    movel([-0.101611, -1.453252, -2.511691, -0.747446, 1.570796, 1.469185],accel_mss,speed_ms,0,blend_radius_m)
    movel([-0.098360, -1.448678, -2.515403, -0.748308, 1.570796, 1.472436],accel_mss,speed_ms,0,blend_radius_m)
    movel([-0.092173, -1.439398, -2.522836, -0.750155, 1.570796, 1.478623],accel_mss,speed_ms,0,blend_radius_m)
    movel([-0.087668, -1.432622, -2.528181, -0.751586, 1.570796, 1.483129],accel_mss,speed_ms,0,blend_radius_m)
    movel([-0.083332, -1.426923, -2.532623, -0.752843, 1.570796, 1.487464],accel_mss,speed_ms,0,blend_radius_m)
    movel([-0.078941, -1.421179, -2.537051, -0.754159, 1.570796, 1.491855],accel_mss,speed_ms,0,blend_radius_m)
    movel([-0.091400, -1.427836, -2.531915, -0.752638, 1.570796, 1.479397],accel_mss,speed_ms,0,blend_radius_m)
    movel([-0.097928, -1.431068, -2.529397, -0.751924, 1.570796, 1.472868],accel_mss,speed_ms,0,blend_radius_m)
    movel([-0.104381, -1.433755, -2.527293, -0.751342, 1.570796, 1.466415],accel_mss,speed_ms,0,blend_radius_m)
    movel([-0.107519, -1.434780, -2.526486, -0.751122, 1.570796, 1.463277],accel_mss,speed_ms,0,blend_radius_m)
    movel([-0.110566, -1.435536, -2.525891, -0.750962, 1.570796, 1.460230],accel_mss,speed_ms,0,blend_radius_m)
    movel([-0.113501, -1.435974, -2.525546, -0.750869, 1.570796, 1.457296],accel_mss,speed_ms,0,blend_radius_m)
    movel([-0.116300, -1.436052, -2.525484, -0.750853, 1.570796, 1.454497],accel_mss,speed_ms,0,blend_radius_m)
    movel([-0.118941, -1.435725, -2.525742, -0.750922, 1.570796, 1.451855],accel_mss,speed_ms,0,blend_radius_m)
    movel([-0.121404, -1.434945, -2.526356, -0.751087, 1.570796, 1.449392],accel_mss,speed_ms,0,blend_radius_m)
    movel([-0.123665, -1.433664, -2.527364, -0.751361, 1.570796, 1.447131],accel_mss,speed_ms,0,blend_radius_m)
    movel([-0.125701, -1.431833, -2.528799, -0.751757, 1.570796, 1.445095],accel_mss,speed_ms,0,blend_radius_m)
    movel([-0.127479, -1.429180, -2.530870, -0.752339, 1.570796, 1.443317],accel_mss,speed_ms,0,blend_radius_m)
    movel([-0.128567, -1.425999, -2.533339, -0.753051, 1.570796, 1.442229],accel_mss,speed_ms,0,blend_radius_m)
    movel([-0.128974, -1.422404, -2.536111, -0.753874, 1.570796, 1.441823],accel_mss,speed_ms,0,blend_radius_m)
    movel([-0.128700, -1.418509, -2.539092, -0.754787, 1.570796, 1.442097],accel_mss,speed_ms,0,blend_radius_m)
    movel([-0.127750, -1.414438, -2.542185, -0.755766, 1.570796, 1.443046],accel_mss,speed_ms,0,blend_radius_m)
    movel([-0.126130, -1.410311, -2.545294, -0.756784, 1.570796, 1.444666],accel_mss,speed_ms,0,blend_radius_m)
    movel([-0.123845, -1.406255, -2.548326, -0.757808, 1.570796, 1.446951],accel_mss,speed_ms,0,blend_radius_m)
    movel([-0.120902, -1.402407, -2.551180, -0.758802, 1.570796, 1.449894],accel_mss,speed_ms,0,blend_radius_m)
    movel([-0.118903, -1.400597, -2.552515, -0.759277, 1.570796, 1.451893],accel_mss,speed_ms,0,blend_radius_m)
    movel([-0.116399, -1.398924, -2.553745, -0.759721, 1.570796, 1.454398],accel_mss,speed_ms,0,blend_radius_m)
    movel([-0.114170, -1.397957, -2.554453, -0.759979, 1.570796, 1.456626],accel_mss,speed_ms,0,blend_radius_m)
    movel([-0.113404, -1.397916, -2.554483, -0.759990, 1.570796, 1.457393],accel_mss,speed_ms,0,blend_radius_m)
    movel([-0.113001, -1.398265, -2.554228, -0.759896, 1.570796, 1.457795],accel_mss,speed_ms,0,blend_radius_m)
    movel([-0.114998, -1.399565, -2.553273, -0.759550, 1.570796, 1.455798],accel_mss,speed_ms,0,blend_radius_m)
    movel([-0.116593, -1.400819, -2.552351, -0.759219, 1.570796, 1.454203],accel_mss,speed_ms,0,blend_radius_m)
    movel([-0.117810, -1.402019, -2.551466, -0.758904, 1.570796, 1.452986],accel_mss,speed_ms,0,blend_radius_m)
    movel([-0.118672, -1.403156, -2.550626, -0.758607, 1.570796, 1.452124],accel_mss,speed_ms,0,blend_radius_m)
    movel([-0.119199, -1.404223, -2.549836, -0.758330, 1.570796, 1.451597],accel_mss,speed_ms,0,blend_radius_m)
    movel([-0.119413, -1.405206, -2.549106, -0.758077, 1.570796, 1.451383],accel_mss,speed_ms,0,blend_radius_m)
    movel([-0.119335, -1.406102, -2.548440, -0.757847, 1.570796, 1.451461],accel_mss,speed_ms,0,blend_radius_m)
    movel([-0.118989, -1.406902, -2.547844, -0.757643, 1.570796, 1.451807],accel_mss,speed_ms,0,blend_radius_m)
    movel([-0.117576, -1.408183, -2.546888, -0.757318, 1.570796, 1.453220],accel_mss,speed_ms,0,blend_radius_m)
    movel([-0.115345, -1.408986, -2.546287, -0.757116, 1.570796, 1.455451],accel_mss,speed_ms,0,blend_radius_m)
    movel([-0.112459, -1.409248, -2.546091, -0.757050, 1.570796, 1.458337],accel_mss,speed_ms,0,blend_radius_m)
    movel([-0.109083, -1.408906, -2.546347, -0.757136, 1.570796, 1.461714],accel_mss,speed_ms,0,blend_radius_m)
    movel([-0.106965, -1.408357, -2.546758, -0.757274, 1.570796, 1.463831],accel_mss,speed_ms,0,blend_radius_m)
    movel([-0.104406, -1.407446, -2.547439, -0.757505, 1.570796, 1.466390],accel_mss,speed_ms,0,blend_radius_m)
    movel([-0.098196, -1.404704, -2.549479, -0.758206, 1.570796, 1.472600],accel_mss,speed_ms,0,blend_radius_m)
    movel([-0.090922, -1.401036, -2.552191, -0.759162, 1.570796, 1.479874],accel_mss,speed_ms,0,blend_radius_m)
    movel([-0.083063, -1.396788, -2.555308, -0.760293, 1.570796, 1.487734],accel_mss,speed_ms,0,blend_radius_m)
    movel([-0.067573, -1.387951, -2.561708, -0.762730, 1.570796, 1.503223],accel_mss,speed_ms,0,blend_radius_m)
    movel([-0.055874, -1.381000, -2.566663, -0.764726, 1.570796, 1.514922],accel_mss,speed_ms,0,blend_radius_m)
    movel([-0.049959, -1.377461, -2.569159, -0.765769, 1.570796, 1.520837],accel_mss,speed_ms,0,blend_radius_m)
    movel([-0.046803, -1.375466, -2.570558, -0.766365, 1.570796, 1.523993],accel_mss,speed_ms,0,blend_radius_m)
    movel([-0.044493, -1.373787, -2.571731, -0.766871, 1.570796, 1.526303],accel_mss,speed_ms,0,blend_radius_m)
    movel([-0.043931, -1.373226, -2.572122, -0.767041, 1.570796, 1.526866],accel_mss,speed_ms,0,blend_radius_m)
    movel([-0.043801, -1.372867, -2.572373, -0.767150, 1.570796, 1.526996],accel_mss,speed_ms,0,blend_radius_m)
    movel([-0.044572, -1.372479, -2.572643, -0.767268, 1.570796, 1.526224],accel_mss,speed_ms,0,blend_radius_m)
    movel([-0.047476, -1.372220, -2.572823, -0.767346, 1.570796, 1.523320],accel_mss,speed_ms,0,blend_radius_m)
    movel([-0.050727, -1.372474, -2.572646, -0.767269, 1.570796, 1.520069],accel_mss,speed_ms,0,blend_radius_m)
    movel([-0.057799, -1.373319, -2.572057, -0.767012, 1.570796, 1.512998],accel_mss,speed_ms,0,blend_radius_m)
    movel([-0.061398, -1.373317, -2.572059, -0.767013, 1.570796, 1.509398],accel_mss,speed_ms,0,blend_radius_m)
    movel([-0.064898, -1.372629, -2.572538, -0.767222, 1.570796, 1.505898],accel_mss,speed_ms,0,blend_radius_m)
    movel([-0.066577, -1.371935, -2.573021, -0.767433, 1.570796, 1.504219],accel_mss,speed_ms,0,blend_radius_m)
    movel([-0.068195, -1.370958, -2.573699, -0.767732, 1.570796, 1.502601],accel_mss,speed_ms,0,blend_radius_m)
    movel([-0.069739, -1.369658, -2.574600, -0.768132, 1.570796, 1.501057],accel_mss,speed_ms,0,blend_radius_m)
    movel([-0.071195, -1.367994, -2.575748, -0.768647, 1.570796, 1.499601],accel_mss,speed_ms,0,blend_radius_m)
    movel([-0.072638, -1.365440, -2.577504, -0.769445, 1.570796, 1.498158],accel_mss,speed_ms,0,blend_radius_m)
    movel([-0.073373, -1.362616, -2.579435, -0.770338, 1.570796, 1.497424],accel_mss,speed_ms,0,blend_radius_m)
    movel([-0.073471, -1.359553, -2.581517, -0.771319, 1.570796, 1.497325],accel_mss,speed_ms,0,blend_radius_m)
    movel([-0.073008, -1.356295, -2.583717, -0.772377, 1.570796, 1.497789],accel_mss,speed_ms,0,blend_radius_m)
    movel([-0.072060, -1.352877, -2.586009, -0.773503, 1.570796, 1.498736],accel_mss,speed_ms,0,blend_radius_m)
    movel([-0.070704, -1.349346, -2.588360, -0.774684, 1.570796, 1.500092],accel_mss,speed_ms,0,blend_radius_m)
    movel([-0.069018, -1.345740, -2.590742, -0.775907, 1.570796, 1.501778],accel_mss,speed_ms,0,blend_radius_m)
    movel([-0.067084, -1.342109, -2.593124, -0.777156, 1.570796, 1.503712],accel_mss,speed_ms,0,blend_radius_m)
    movel([-0.062875, -1.335380, -2.597489, -0.779519, 1.570796, 1.507922],accel_mss,speed_ms,0,blend_radius_m)
    movel([-0.058564, -1.329688, -2.601135, -0.781566, 1.570796, 1.512232],accel_mss,speed_ms,0,blend_radius_m)
    movel([-0.054523, -1.325129, -2.604023, -0.783238, 1.570796, 1.516273],accel_mss,speed_ms,0,blend_radius_m)
    movel([-0.051129, -1.321798, -2.606115, -0.784476, 1.570796, 1.519667],accel_mss,speed_ms,0,blend_radius_m)
    movel([-0.045692, -1.317282, -2.608929, -0.786179, 1.570796, 1.525104],accel_mss,speed_ms,0,blend_radius_m)
    movel([-0.040005, -1.313397, -2.611327, -0.787665, 1.570796, 1.530791],accel_mss,speed_ms,0,blend_radius_m)
    movel([-0.034153, -1.310170, -2.613304, -0.788914, 1.570796, 1.536643],accel_mss,speed_ms,0,blend_radius_m)
    movel([-0.028236, -1.307628, -2.614852, -0.789908, 1.570796, 1.542561],accel_mss,speed_ms,0,blend_radius_m)
    movel([-0.022348, -1.305795, -2.615963, -0.790631, 1.570796, 1.548449],accel_mss,speed_ms,0,blend_radius_m)
    movel([-0.016580, -1.304686, -2.616634, -0.791070, 1.570796, 1.554216],accel_mss,speed_ms,0,blend_radius_m)
    movel([-0.011030, -1.304317, -2.616856, -0.791216, 1.570796, 1.559766],accel_mss,speed_ms,0,blend_radius_m)
    movel([-0.005791, -1.304700, -2.616625, -0.791064, 1.570796, 1.565005],accel_mss,speed_ms,0,blend_radius_m)
    movel([-0.001418, -1.305694, -2.616024, -0.790670, 1.570796, 1.569378],accel_mss,speed_ms,0,blend_radius_m)
    movel([0.002673, -1.307080, -2.615185, -0.790124, 1.570796, 1.573469],accel_mss,speed_ms,0,blend_radius_m)
    movel([0.006644, -1.308526, -2.614306, -0.789556, 1.570796, 1.577440],accel_mss,speed_ms,0,blend_radius_m)
    movel([0.010668, -1.309702, -2.613590, -0.789097, 1.570796, 1.581464],accel_mss,speed_ms,0,blend_radius_m)
    movel([0.014918, -1.310286, -2.613234, -0.788870, 1.570796, 1.585715],accel_mss,speed_ms,0,blend_radius_m)
    movel([0.017183, -1.310251, -2.613255, -0.788883, 1.570796, 1.587979],accel_mss,speed_ms,0,blend_radius_m)
    movel([0.019570, -1.309949, -2.613439, -0.789001, 1.570796, 1.590366],accel_mss,speed_ms,0,blend_radius_m)
    movel([0.022104, -1.309335, -2.613814, -0.789240, 1.570796, 1.592900],accel_mss,speed_ms,0,blend_radius_m)
    movel([0.024809, -1.308369, -2.614402, -0.789618, 1.570796, 1.595605],accel_mss,speed_ms,0,blend_radius_m)
    movel([0.027712, -1.307006, -2.615230, -0.790153, 1.570796, 1.598508],accel_mss,speed_ms,0,blend_radius_m)
    movel([0.030836, -1.305204, -2.616321, -0.790864, 1.570796, 1.601633],accel_mss,speed_ms,0,blend_radius_m)
    movel([0.033462, -1.303311, -2.617462, -0.791616, 1.570796, 1.604259],accel_mss,speed_ms,0,blend_radius_m)
    movel([0.035502, -1.301346, -2.618642, -0.792401, 1.570796, 1.606298],accel_mss,speed_ms,0,blend_radius_m)
    movel([0.036986, -1.299357, -2.619831, -0.793201, 1.570796, 1.607782],accel_mss,speed_ms,0,blend_radius_m)
    movel([0.037958, -1.297392, -2.621001, -0.793996, 1.570796, 1.608754],accel_mss,speed_ms,0,blend_radius_m)
    movel([0.038450, -1.295502, -2.622121, -0.794766, 1.570796, 1.609246],accel_mss,speed_ms,0,blend_radius_m)
    movel([0.038495, -1.293743, -2.623160, -0.795486, 1.570796, 1.609292],accel_mss,speed_ms,0,blend_radius_m)
    movel([0.038134, -1.292163, -2.624089, -0.796137, 1.570796, 1.608931],accel_mss,speed_ms,0,blend_radius_m)
    movel([0.037403, -1.290817, -2.624879, -0.796693, 1.570796, 1.608199],accel_mss,speed_ms,0,blend_radius_m)
    movel([0.036339, -1.289760, -2.625497, -0.797132, 1.570796, 1.607135],accel_mss,speed_ms,0,blend_radius_m)
    movel([0.034980, -1.289045, -2.625915, -0.797429, 1.570796, 1.605776],accel_mss,speed_ms,0,blend_radius_m)
    movel([0.033366, -1.288725, -2.626101, -0.797563, 1.570796, 1.604163],accel_mss,speed_ms,0,blend_radius_m)
    movel([0.031539, -1.288853, -2.626027, -0.797510, 1.570796, 1.602335],accel_mss,speed_ms,0,blend_radius_m)
    movel([0.029539, -1.289474, -2.625664, -0.797251, 1.570796, 1.600335],accel_mss,speed_ms,0,blend_radius_m)
    movel([0.027413, -1.290642, -2.624982, -0.796766, 1.570796, 1.598209],accel_mss,speed_ms,0,blend_radius_m)
    movel([0.025201, -1.292403, -2.623948, -0.796037, 1.570796, 1.595998],accel_mss,speed_ms,0,blend_radius_m)
    movel([0.022949, -1.294798, -2.622537, -0.795054, 1.570796, 1.593746],accel_mss,speed_ms,0,blend_radius_m)
    movel([0.024835, -1.294234, -2.622870, -0.795285, 1.570796, 1.595631],accel_mss,speed_ms,0,blend_radius_m)
    movel([0.026385, -1.294077, -2.622963, -0.795349, 1.570796, 1.597182],accel_mss,speed_ms,0,blend_radius_m)
    movel([0.027564, -1.294304, -2.622829, -0.795256, 1.570796, 1.598361],accel_mss,speed_ms,0,blend_radius_m)
    movel([0.028342, -1.294888, -2.622484, -0.795017, 1.570796, 1.599138],accel_mss,speed_ms,0,blend_radius_m)
    movel([0.028683, -1.295809, -2.621940, -0.794641, 1.570796, 1.599479],accel_mss,speed_ms,0,blend_radius_m)
    movel([0.028557, -1.297039, -2.621210, -0.794140, 1.570796, 1.599354],accel_mss,speed_ms,0,blend_radius_m)
    movel([0.027935, -1.298550, -2.620312, -0.793527, 1.570796, 1.598731],accel_mss,speed_ms,0,blend_radius_m)
    movel([0.026784, -1.300320, -2.619256, -0.792813, 1.570796, 1.597581],accel_mss,speed_ms,0,blend_radius_m)
    movel([0.024280, -1.303118, -2.617578, -0.791693, 1.570796, 1.595077],accel_mss,speed_ms,0,blend_radius_m)
    movel([0.021602, -1.305191, -2.616329, -0.790870, 1.570796, 1.592398],accel_mss,speed_ms,0,blend_radius_m)
    movel([0.018815, -1.306593, -2.615480, -0.790316, 1.570796, 1.589612],accel_mss,speed_ms,0,blend_radius_m)
    movel([0.016000, -1.307372, -2.615008, -0.790009, 1.570796, 1.586796],accel_mss,speed_ms,0,blend_radius_m)
    movel([0.013225, -1.307572, -2.614887, -0.789931, 1.570796, 1.584021],accel_mss,speed_ms,0,blend_radius_m)
    movel([0.010566, -1.307233, -2.615092, -0.790064, 1.570796, 1.581362],accel_mss,speed_ms,0,blend_radius_m)
    movel([0.008102, -1.306397, -2.615599, -0.790393, 1.570796, 1.578898],accel_mss,speed_ms,0,blend_radius_m)
    movel([0.005906, -1.305103, -2.616381, -0.790904, 1.570796, 1.576702],accel_mss,speed_ms,0,blend_radius_m)
    movel([0.004062, -1.303381, -2.617420, -0.791588, 1.570796, 1.574859],accel_mss,speed_ms,0,blend_radius_m)
    movel([0.002647, -1.301272, -2.618686, -0.792431, 1.570796, 1.573443],accel_mss,speed_ms,0,blend_radius_m)
    movel([0.001748, -1.298803, -2.620161, -0.793425, 1.570796, 1.572545],accel_mss,speed_ms,0,blend_radius_m)
    movel([0.001450, -1.296012, -2.621819, -0.794558, 1.570796, 1.572246],accel_mss,speed_ms,0,blend_radius_m)
    movel([0.001841, -1.292927, -2.623641, -0.795822, 1.570796, 1.572637],accel_mss,speed_ms,0,blend_radius_m)
    movel([0.003010, -1.289582, -2.625601, -0.797206, 1.570796, 1.573806],accel_mss,speed_ms,0,blend_radius_m)
    movel([0.005052, -1.286011, -2.627679, -0.798699, 1.570796, 1.575848],accel_mss,speed_ms,0,blend_radius_m)
    movel([0.008055, -1.282252, -2.629848, -0.800289, 1.570796, 1.578851],accel_mss,speed_ms,0,blend_radius_m)
    movel([0.010545, -1.279696, -2.631313, -0.801380, 1.570796, 1.581341],accel_mss,speed_ms,0,blend_radius_m)
    movel([0.013182, -1.277305, -2.632676, -0.802408, 1.570796, 1.583978],accel_mss,speed_ms,0,blend_radius_m)
    movel([0.015934, -1.275092, -2.633932, -0.803365, 1.570796, 1.586731],accel_mss,speed_ms,0,blend_radius_m)
    movel([0.018783, -1.273077, -2.635069, -0.804243, 1.570796, 1.589579],accel_mss,speed_ms,0,blend_radius_m)
    movel([0.021695, -1.271275, -2.636082, -0.805032, 1.570796, 1.592491],accel_mss,speed_ms,0,blend_radius_m)
    movel([0.024648, -1.269703, -2.636963, -0.805723, 1.570796, 1.595444],accel_mss,speed_ms,0,blend_radius_m)
    movel([0.027613, -1.268378, -2.637703, -0.806308, 1.570796, 1.598410],accel_mss,speed_ms,0,blend_radius_m)
    movel([0.030563, -1.267314, -2.638295, -0.806780, 1.570796, 1.601360],accel_mss,speed_ms,0,blend_radius_m)
    movel([0.033469, -1.266531, -2.638731, -0.807128, 1.570796, 1.604266],accel_mss,speed_ms,0,blend_radius_m)
    movel([0.036305, -1.266038, -2.639004, -0.807347, 1.570796, 1.607101],accel_mss,speed_ms,0,blend_radius_m)
    movel([0.039042, -1.265856, -2.639105, -0.807428, 1.570796, 1.609838],accel_mss,speed_ms,0,blend_radius_m)
    movel([0.041654, -1.265996, -2.639027, -0.807366, 1.570796, 1.612451],accel_mss,speed_ms,0,blend_radius_m)
    movel([0.044111, -1.266472, -2.638763, -0.807154, 1.570796, 1.614907],accel_mss,speed_ms,0,blend_radius_m)
    movel([0.046390, -1.267293, -2.638307, -0.806789, 1.570796, 1.617186],accel_mss,speed_ms,0,blend_radius_m)
    movel([0.048461, -1.268477, -2.637648, -0.806264, 1.570796, 1.619257],accel_mss,speed_ms,0,blend_radius_m)
    movel([0.050299, -1.270031, -2.636779, -0.805578, 1.570796, 1.621095],accel_mss,speed_ms,0,blend_radius_m)
    movel([0.051489, -1.272144, -2.635594, -0.804650, 1.570796, 1.622286],accel_mss,speed_ms,0,blend_radius_m)
    movel([0.052205, -1.274852, -2.634067, -0.803469, 1.570796, 1.623002],accel_mss,speed_ms,0,blend_radius_m)
    movel([0.052659, -1.277284, -2.632688, -0.802416, 1.570796, 1.623456],accel_mss,speed_ms,0,blend_radius_m)
    movel([0.053064, -1.278582, -2.631949, -0.801858, 1.570796, 1.623860],accel_mss,speed_ms,0,blend_radius_m)
    movel([0.054264, -1.278779, -2.631837, -0.801773, 1.570796, 1.625060],accel_mss,speed_ms,0,blend_radius_m)
    movel([0.056461, -1.278666, -2.631901, -0.801821, 1.570796, 1.627257],accel_mss,speed_ms,0,blend_radius_m)
    movel([0.058885, -1.278544, -2.631971, -0.801874, 1.570796, 1.629681],accel_mss,speed_ms,0,blend_radius_m)
    movel([0.060765, -1.278700, -2.631882, -0.801807, 1.570796, 1.631562],accel_mss,speed_ms,0,blend_radius_m)
    movel([0.062834, -1.279532, -2.631407, -0.801450, 1.570796, 1.633631],accel_mss,speed_ms,0,blend_radius_m)
    movel([0.064472, -1.280680, -2.630751, -0.800959, 1.570796, 1.635268],accel_mss,speed_ms,0,blend_radius_m)
    movel([0.065692, -1.282108, -2.629931, -0.800350, 1.570796, 1.636488],accel_mss,speed_ms,0,blend_radius_m)
    movel([0.066513, -1.283776, -2.628971, -0.799642, 1.570796, 1.637309],accel_mss,speed_ms,0,blend_radius_m)
    movel([0.066955, -1.285648, -2.627889, -0.798852, 1.570796, 1.637752],accel_mss,speed_ms,0,blend_radius_m)
    movel([0.067036, -1.287682, -2.626708, -0.797998, 1.570796, 1.637832],accel_mss,speed_ms,0,blend_radius_m)
    movel([0.066776, -1.289843, -2.625448, -0.797097, 1.570796, 1.637572],accel_mss,speed_ms,0,blend_radius_m)
    movel([0.066191, -1.292094, -2.624130, -0.796165, 1.570796, 1.636988],accel_mss,speed_ms,0,blend_radius_m)
    movel([0.065300, -1.294401, -2.622772, -0.795216, 1.570796, 1.636097],accel_mss,speed_ms,0,blend_radius_m)
    movel([0.064122, -1.296725, -2.621397, -0.794267, 1.570796, 1.634918],accel_mss,speed_ms,0,blend_radius_m)
    movel([0.062673, -1.299035, -2.620023, -0.793331, 1.570796, 1.633469],accel_mss,speed_ms,0,blend_radius_m)
    speed_ms = 0.003
    movel([0.062673, -1.292173, -2.616738, -0.803478, 1.570796, 1.633469],accel_mss,speed_ms,0,blend_radius_m)
    speed_ms = 0.05
    movel([0.062673, -1.265901, -2.603322, -0.843166, 1.570796, 1.633469],accel_mss,speed_ms,0,blend_radius_m)
    #M_RunCode9
    movel([0.079276, -1.257744, -2.607923, -0.846722, 1.570796, 1.650073],accel_mss,speed_ms,0,blend_radius_m)
    #M_RunCode3
    movel([0.079276, -1.284127, -2.621447, -0.806816, 1.570796, 1.650073],accel_mss,speed_ms,0,blend_radius_m)
    speed_ms = 0.003
    movel([0.079276, -1.291022, -2.624759, -0.796608, 1.570796, 1.650073],accel_mss,speed_ms,0,blend_radius_m)
    speed_ms = 0.02
    movel([0.079182, -1.289313, -2.625758, -0.797318, 1.570796, 1.649979],accel_mss,speed_ms,0,blend_radius_m)
    movel([0.079578, -1.285585, -2.627926, -0.798879, 1.570796, 1.650374],accel_mss,speed_ms,0,blend_radius_m)
    movel([0.079753, -1.282031, -2.629975, -0.800383, 1.570796, 1.650549],accel_mss,speed_ms,0,blend_radius_m)
    movel([0.079381, -1.280546, -2.630827, -0.801016, 1.570796, 1.650178],accel_mss,speed_ms,0,blend_radius_m)
    movel([0.078497, -1.279378, -2.631495, -0.801516, 1.570796, 1.649293],accel_mss,speed_ms,0,blend_radius_m)
    movel([0.079533, -1.279857, -2.631221, -0.801311, 1.570796, 1.650329],accel_mss,speed_ms,0,blend_radius_m)
    movel([0.081004, -1.281148, -2.630482, -0.800759, 1.570796, 1.651801],accel_mss,speed_ms,0,blend_radius_m)
    movel([0.081818, -1.282779, -2.629545, -0.800065, 1.570796, 1.652614],accel_mss,speed_ms,0,blend_radius_m)
    movel([0.082178, -1.284645, -2.628469, -0.799275, 1.570796, 1.652974],accel_mss,speed_ms,0,blend_radius_m)
    movel([0.082289, -1.286641, -2.627313, -0.798435, 1.570796, 1.653085],accel_mss,speed_ms,0,blend_radius_m)
    movel([0.082574, -1.290622, -2.624993, -0.796774, 1.570796, 1.653370],accel_mss,speed_ms,0,blend_radius_m)
    movel([0.083146, -1.292412, -2.623943, -0.796034, 1.570796, 1.653942],accel_mss,speed_ms,0,blend_radius_m)
    movel([0.084268, -1.293936, -2.623046, -0.795407, 1.570796, 1.655064],accel_mss,speed_ms,0,blend_radius_m)
    movel([0.086018, -1.295241, -2.622276, -0.794873, 1.570796, 1.656814],accel_mss,speed_ms,0,blend_radius_m)
    movel([0.087065, -1.295825, -2.621930, -0.794634, 1.570796, 1.657861],accel_mss,speed_ms,0,blend_radius_m)
    movel([0.087819, -1.295990, -2.621832, -0.794567, 1.570796, 1.658615],accel_mss,speed_ms,0,blend_radius_m)
    movel([0.089062, -1.295029, -2.622401, -0.794959, 1.570796, 1.659858],accel_mss,speed_ms,0,blend_radius_m)
    movel([0.090104, -1.294278, -2.622844, -0.795267, 1.570796, 1.660900],accel_mss,speed_ms,0,blend_radius_m)
    movel([0.091245, -1.293667, -2.623204, -0.795517, 1.570796, 1.662041],accel_mss,speed_ms,0,blend_radius_m)
    movel([0.093544, -1.292886, -2.623664, -0.795839, 1.570796, 1.664341],accel_mss,speed_ms,0,blend_radius_m)
    movel([0.095252, -1.292611, -2.623826, -0.795952, 1.570796, 1.666049],accel_mss,speed_ms,0,blend_radius_m)
    movel([0.096505, -1.292746, -2.623747, -0.795896, 1.570796, 1.667301],accel_mss,speed_ms,0,blend_radius_m)
    movel([0.097444, -1.293201, -2.623479, -0.795709, 1.570796, 1.668240],accel_mss,speed_ms,0,blend_radius_m)
    movel([0.098946, -1.294696, -2.622598, -0.795095, 1.570796, 1.669743],accel_mss,speed_ms,0,blend_radius_m)
    movel([0.100895, -1.296364, -2.621610, -0.794414, 1.570796, 1.671692],accel_mss,speed_ms,0,blend_radius_m)
    movel([0.104110, -1.298008, -2.620635, -0.793747, 1.570796, 1.674906],accel_mss,speed_ms,0,blend_radius_m)
    movel([0.107423, -1.299511, -2.619739, -0.793139, 1.570796, 1.678219],accel_mss,speed_ms,0,blend_radius_m)
    movel([0.110560, -1.301203, -2.618727, -0.792458, 1.570796, 1.681356],accel_mss,speed_ms,0,blend_radius_m)
    movel([0.113253, -1.303396, -2.617411, -0.791582, 1.570796, 1.684050],accel_mss,speed_ms,0,blend_radius_m)
    movel([0.114384, -1.304882, -2.616515, -0.790992, 1.570796, 1.685180],accel_mss,speed_ms,0,blend_radius_m)
    movel([0.115256, -1.306555, -2.615503, -0.790331, 1.570796, 1.686053],accel_mss,speed_ms,0,blend_radius_m)
    movel([0.116468, -1.310252, -2.613254, -0.788883, 1.570796, 1.687264],accel_mss,speed_ms,0,blend_radius_m)
    movel([0.117372, -1.314078, -2.610908, -0.787403, 1.570796, 1.688168],accel_mss,speed_ms,0,blend_radius_m)
    movel([0.118449, -1.317628, -2.608714, -0.786047, 1.570796, 1.689246],accel_mss,speed_ms,0,blend_radius_m)
    movel([0.121104, -1.322927, -2.605407, -0.784054, 1.570796, 1.691901],accel_mss,speed_ms,0,blend_radius_m)
    movel([0.122316, -1.325141, -2.604015, -0.783233, 1.570796, 1.693112],accel_mss,speed_ms,0,blend_radius_m)
    movel([0.123257, -1.327360, -2.602613, -0.782416, 1.570796, 1.694054],accel_mss,speed_ms,0,blend_radius_m)
    movel([0.123798, -1.329795, -2.601066, -0.781528, 1.570796, 1.694594],accel_mss,speed_ms,0,blend_radius_m)
    movel([0.123793, -1.332661, -2.599236, -0.780492, 1.570796, 1.694590],accel_mss,speed_ms,0,blend_radius_m)
    movel([0.123109, -1.336167, -2.596982, -0.779240, 1.570796, 1.693905],accel_mss,speed_ms,0,blend_radius_m)
    movel([0.121617, -1.340512, -2.594165, -0.777711, 1.570796, 1.692413],accel_mss,speed_ms,0,blend_radius_m)
    movel([0.120010, -1.344054, -2.591850, -0.776485, 1.570796, 1.690807],accel_mss,speed_ms,0,blend_radius_m)
    movel([0.118181, -1.347275, -2.589730, -0.775384, 1.570796, 1.688977],accel_mss,speed_ms,0,blend_radius_m)
    movel([0.116146, -1.350191, -2.587799, -0.774399, 1.570796, 1.686942],accel_mss,speed_ms,0,blend_radius_m)
    movel([0.113919, -1.352822, -2.586045, -0.773521, 1.570796, 1.684715],accel_mss,speed_ms,0,blend_radius_m)
    movel([0.111524, -1.355182, -2.584465, -0.772742, 1.570796, 1.682320],accel_mss,speed_ms,0,blend_radius_m)
    movel([0.108974, -1.357288, -2.583048, -0.772053, 1.570796, 1.679770],accel_mss,speed_ms,0,blend_radius_m)
    movel([0.106287, -1.359152, -2.581788, -0.771448, 1.570796, 1.677084],accel_mss,speed_ms,0,blend_radius_m)
    movel([0.103479, -1.360792, -2.580676, -0.770920, 1.570796, 1.674275],accel_mss,speed_ms,0,blend_radius_m)
    movel([0.100570, -1.362219, -2.579706, -0.770464, 1.570796, 1.671366],accel_mss,speed_ms,0,blend_radius_m)
    movel([0.097571, -1.363450, -2.578866, -0.770073, 1.570796, 1.668367],accel_mss,speed_ms,0,blend_radius_m)
    movel([0.091375, -1.365371, -2.577552, -0.769466, 1.570796, 1.662171],accel_mss,speed_ms,0,blend_radius_m)
    movel([0.085030, -1.366656, -2.576669, -0.769064, 1.570796, 1.655826],accel_mss,speed_ms,0,blend_radius_m)
    movel([0.078670, -1.367404, -2.576155, -0.768830, 1.570796, 1.649466],accel_mss,speed_ms,0,blend_radius_m)
    movel([0.072831, -1.367616, -2.576008, -0.768764, 1.570796, 1.643627],accel_mss,speed_ms,0,blend_radius_m)
    movel([0.065389, -1.367790, -2.575889, -0.768710, 1.570796, 1.636186],accel_mss,speed_ms,0,blend_radius_m)
    movel([0.057017, -1.368376, -2.575485, -0.768528, 1.570796, 1.627813],accel_mss,speed_ms,0,blend_radius_m)
    movel([0.052698, -1.368956, -2.575085, -0.768348, 1.570796, 1.623495],accel_mss,speed_ms,0,blend_radius_m)
    movel([0.048406, -1.369796, -2.574504, -0.768089, 1.570796, 1.619202],accel_mss,speed_ms,0,blend_radius_m)
    movel([0.044238, -1.370942, -2.573710, -0.767737, 1.570796, 1.615034],accel_mss,speed_ms,0,blend_radius_m)
    movel([0.040279, -1.372440, -2.572669, -0.767279, 1.570796, 1.611075],accel_mss,speed_ms,0,blend_radius_m)
    movel([0.036623, -1.374335, -2.571349, -0.766705, 1.570796, 1.607420],accel_mss,speed_ms,0,blend_radius_m)
    movel([0.033366, -1.376665, -2.569718, -0.766006, 1.570796, 1.604162],accel_mss,speed_ms,0,blend_radius_m)
    movel([0.031912, -1.378007, -2.568775, -0.765607, 1.570796, 1.602708],accel_mss,speed_ms,0,blend_radius_m)
    movel([0.030592, -1.379474, -2.567741, -0.765174, 1.570796, 1.601389],accel_mss,speed_ms,0,blend_radius_m)
    movel([0.029416, -1.381068, -2.566615, -0.764706, 1.570796, 1.600212],accel_mss,speed_ms,0,blend_radius_m)
    movel([0.028394, -1.382796, -2.565389, -0.764204, 1.570796, 1.599190],accel_mss,speed_ms,0,blend_radius_m)
    movel([0.027538, -1.384663, -2.564061, -0.763666, 1.570796, 1.598334],accel_mss,speed_ms,0,blend_radius_m)
    movel([0.026856, -1.386673, -2.562624, -0.763092, 1.570796, 1.597652],accel_mss,speed_ms,0,blend_radius_m)
    movel([0.026061, -1.391141, -2.559411, -0.761837, 1.570796, 1.596857],accel_mss,speed_ms,0,blend_radius_m)
    movel([0.026322, -1.393089, -2.558001, -0.761299, 1.570796, 1.597118],accel_mss,speed_ms,0,blend_radius_m)
    movel([0.027050, -1.394855, -2.556718, -0.760816, 1.570796, 1.597846],accel_mss,speed_ms,0,blend_radius_m)
    movel([0.028269, -1.396415, -2.555581, -0.760393, 1.570796, 1.599066],accel_mss,speed_ms,0,blend_radius_m)
    movel([0.029998, -1.397736, -2.554615, -0.760038, 1.570796, 1.600794],accel_mss,speed_ms,0,blend_radius_m)
    movel([0.031257, -1.394714, -2.556821, -0.760855, 1.570796, 1.602054],accel_mss,speed_ms,0,blend_radius_m)
    movel([0.032818, -1.391796, -2.558938, -0.761656, 1.570796, 1.603614],accel_mss,speed_ms,0,blend_radius_m)
    movel([0.034657, -1.389000, -2.560954, -0.762435, 1.570796, 1.605453],accel_mss,speed_ms,0,blend_radius_m)
    movel([0.036750, -1.386344, -2.562860, -0.763185, 1.570796, 1.607546],accel_mss,speed_ms,0,blend_radius_m)
    movel([0.039067, -1.383848, -2.564641, -0.763900, 1.570796, 1.609864],accel_mss,speed_ms,0,blend_radius_m)
    movel([0.041589, -1.381528, -2.566289, -0.764572, 1.570796, 1.612385],accel_mss,speed_ms,0,blend_radius_m)
    movel([0.044286, -1.379407, -2.567789, -0.765193, 1.570796, 1.615082],accel_mss,speed_ms,0,blend_radius_m)
    movel([0.047131, -1.377502, -2.569130, -0.765757, 1.570796, 1.617927],accel_mss,speed_ms,0,blend_radius_m)
    movel([0.050098, -1.375832, -2.570302, -0.766255, 1.570796, 1.620894],accel_mss,speed_ms,0,blend_radius_m)
    movel([0.053153, -1.374420, -2.571289, -0.766679, 1.570796, 1.623949],accel_mss,speed_ms,0,blend_radius_m)
    movel([0.056273, -1.373281, -2.572084, -0.767024, 1.570796, 1.627069],accel_mss,speed_ms,0,blend_radius_m)
    movel([0.059427, -1.372434, -2.572674, -0.767281, 1.570796, 1.630223],accel_mss,speed_ms,0,blend_radius_m)
    movel([0.062582, -1.371902, -2.573043, -0.767443, 1.570796, 1.633378],accel_mss,speed_ms,0,blend_radius_m)
    movel([0.065712, -1.371700, -2.573184, -0.767505, 1.570796, 1.636508],accel_mss,speed_ms,0,blend_radius_m)
    movel([0.068788, -1.371845, -2.573083, -0.767461, 1.570796, 1.639584],accel_mss,speed_ms,0,blend_radius_m)
    movel([0.071774, -1.372351, -2.572731, -0.767306, 1.570796, 1.642571],accel_mss,speed_ms,0,blend_radius_m)
    movel([0.074076, -1.373042, -2.572251, -0.767097, 1.570796, 1.644873],accel_mss,speed_ms,0,blend_radius_m)
    movel([0.076126, -1.373943, -2.571622, -0.766823, 1.570796, 1.646923],accel_mss,speed_ms,0,blend_radius_m)
    movel([0.077925, -1.375042, -2.570854, -0.766492, 1.570796, 1.648722],accel_mss,speed_ms,0,blend_radius_m)
    movel([0.079482, -1.376320, -2.569960, -0.766109, 1.570796, 1.650279],accel_mss,speed_ms,0,blend_radius_m)
    movel([0.081892, -1.379341, -2.567836, -0.765213, 1.570796, 1.652688],accel_mss,speed_ms,0,blend_radius_m)
    movel([0.083393, -1.382869, -2.565338, -0.764183, 1.570796, 1.654189],accel_mss,speed_ms,0,blend_radius_m)
    movel([0.084042, -1.386769, -2.562555, -0.763064, 1.570796, 1.654838],accel_mss,speed_ms,0,blend_radius_m)
    movel([0.083884, -1.390908, -2.559579, -0.761902, 1.570796, 1.654680],accel_mss,speed_ms,0,blend_radius_m)
    movel([0.082968, -1.395161, -2.556495, -0.760733, 1.570796, 1.653765],accel_mss,speed_ms,0,blend_radius_m)
    movel([0.081349, -1.399402, -2.553394, -0.759594, 1.570796, 1.652145],accel_mss,speed_ms,0,blend_radius_m)
    movel([0.079067, -1.403514, -2.550361, -0.758514, 1.570796, 1.649863],accel_mss,speed_ms,0,blend_radius_m)
    movel([0.076168, -1.407383, -2.547485, -0.757521, 1.570796, 1.646964],accel_mss,speed_ms,0,blend_radius_m)
    movel([0.072694, -1.410900, -2.544852, -0.756637, 1.570796, 1.643491],accel_mss,speed_ms,0,blend_radius_m)
    movel([0.070752, -1.412493, -2.543653, -0.756243, 1.570796, 1.641548],accel_mss,speed_ms,0,blend_radius_m)
    movel([0.068679, -1.413959, -2.542547, -0.755883, 1.570796, 1.639476],accel_mss,speed_ms,0,blend_radius_m)
    movel([0.066479, -1.415283, -2.541545, -0.755561, 1.570796, 1.637275],accel_mss,speed_ms,0,blend_radius_m)
    movel([0.064155, -1.416455, -2.540656, -0.755278, 1.570796, 1.634951],accel_mss,speed_ms,0,blend_radius_m)
    movel([0.061709, -1.417461, -2.539891, -0.755037, 1.570796, 1.632505],accel_mss,speed_ms,0,blend_radius_m)
    movel([0.059146, -1.418290, -2.539259, -0.754840, 1.570796, 1.629943],accel_mss,speed_ms,0,blend_radius_m)
    movel([0.056468, -1.418926, -2.538774, -0.754689, 1.570796, 1.627265],accel_mss,speed_ms,0,blend_radius_m)
    movel([0.053678, -1.419360, -2.538443, -0.754586, 1.570796, 1.624474],accel_mss,speed_ms,0,blend_radius_m)
    movel([0.050775, -1.419580, -2.538275, -0.754534, 1.570796, 1.621571],accel_mss,speed_ms,0,blend_radius_m)
    movel([0.047763, -1.419572, -2.538281, -0.754536, 1.570796, 1.618560],accel_mss,speed_ms,0,blend_radius_m)
    movel([0.045463, -1.419231, -2.538541, -0.754617, 1.570796, 1.616260],accel_mss,speed_ms,0,blend_radius_m)
    movel([0.039389, -1.417785, -2.539644, -0.754960, 1.570796, 1.610185],accel_mss,speed_ms,0,blend_radius_m)
    movel([0.035310, -1.416454, -2.540656, -0.755279, 1.570796, 1.606106],accel_mss,speed_ms,0,blend_radius_m)
    movel([0.030735, -1.414611, -2.542054, -0.755724, 1.570796, 1.601531],accel_mss,speed_ms,0,blend_radius_m)
    movel([0.025805, -1.412176, -2.543892, -0.756321, 1.570796, 1.596601],accel_mss,speed_ms,0,blend_radius_m)
    movel([0.020668, -1.409061, -2.546231, -0.757097, 1.570796, 1.591464],accel_mss,speed_ms,0,blend_radius_m)
    movel([0.017364, -1.406564, -2.548096, -0.757729, 1.570796, 1.588160],accel_mss,speed_ms,0,blend_radius_m)
    movel([0.014706, -1.403978, -2.550018, -0.758394, 1.570796, 1.585503],accel_mss,speed_ms,0,blend_radius_m)
    movel([0.012640, -1.401332, -2.551973, -0.759084, 1.570796, 1.583436],accel_mss,speed_ms,0,blend_radius_m)
    movel([0.011109, -1.398658, -2.553940, -0.759792, 1.570796, 1.581905],accel_mss,speed_ms,0,blend_radius_m)
    movel([0.010057, -1.395981, -2.555897, -0.760510, 1.570796, 1.580853],accel_mss,speed_ms,0,blend_radius_m)
    movel([0.009421, -1.393343, -2.557817, -0.761229, 1.570796, 1.580217],accel_mss,speed_ms,0,blend_radius_m)
    movel([0.009147, -1.390773, -2.559676, -0.761939, 1.570796, 1.579944],accel_mss,speed_ms,0,blend_radius_m)
    movel([0.009172, -1.388310, -2.561450, -0.762629, 1.570796, 1.579968],accel_mss,speed_ms,0,blend_radius_m)
    movel([0.009872, -1.383854, -2.564637, -0.763898, 1.570796, 1.580668],accel_mss,speed_ms,0,blend_radius_m)
    movel([0.011015, -1.380280, -2.567172, -0.764937, 1.570796, 1.581812],accel_mss,speed_ms,0,blend_radius_m)
    movel([0.012088, -1.377904, -2.568847, -0.765637, 1.570796, 1.582885],accel_mss,speed_ms,0,blend_radius_m)
    movel([0.012563, -1.377043, -2.569453, -0.765893, 1.570796, 1.583360],accel_mss,speed_ms,0,blend_radius_m)
    movel([0.015106, -1.373061, -2.572237, -0.767091, 1.570796, 1.585902],accel_mss,speed_ms,0,blend_radius_m)
    movel([0.017908, -1.369437, -2.574752, -0.768200, 1.570796, 1.588704],accel_mss,speed_ms,0,blend_radius_m)
    movel([0.020922, -1.366164, -2.577007, -0.769218, 1.570796, 1.591718],accel_mss,speed_ms,0,blend_radius_m)
    movel([0.024100, -1.363226, -2.579019, -0.770144, 1.570796, 1.594896],accel_mss,speed_ms,0,blend_radius_m)
    movel([0.027388, -1.360613, -2.580798, -0.770978, 1.570796, 1.598185],accel_mss,speed_ms,0,blend_radius_m)
    movel([0.030737, -1.358314, -2.582355, -0.771720, 1.570796, 1.601534],accel_mss,speed_ms,0,blend_radius_m)
    movel([0.034100, -1.356306, -2.583709, -0.772374, 1.570796, 1.604897],accel_mss,speed_ms,0,blend_radius_m)
    movel([0.037421, -1.354581, -2.584868, -0.772940, 1.570796, 1.608218],accel_mss,speed_ms,0,blend_radius_m)
    movel([0.043743, -1.351902, -2.586660, -0.773827, 1.570796, 1.614539],accel_mss,speed_ms,0,blend_radius_m)
    movel([0.049305, -1.350125, -2.587843, -0.774422, 1.570796, 1.620101],accel_mss,speed_ms,0,blend_radius_m)
    movel([0.053716, -1.349086, -2.588532, -0.774771, 1.570796, 1.624512],accel_mss,speed_ms,0,blend_radius_m)
    movel([0.056596, -1.348614, -2.588845, -0.774930, 1.570796, 1.627392],accel_mss,speed_ms,0,blend_radius_m)
    movel([0.063455, -1.347440, -2.589622, -0.775328, 1.570796, 1.634252],accel_mss,speed_ms,0,blend_radius_m)
    movel([0.070821, -1.346624, -2.590160, -0.775605, 1.570796, 1.641617],accel_mss,speed_ms,0,blend_radius_m)
    movel([0.078298, -1.345957, -2.590600, -0.775832, 1.570796, 1.649094],accel_mss,speed_ms,0,blend_radius_m)
    movel([0.085507, -1.345214, -2.591089, -0.776087, 1.570796, 1.656303],accel_mss,speed_ms,0,blend_radius_m)
    movel([0.092080, -1.344157, -2.591783, -0.776449, 1.570796, 1.662876],accel_mss,speed_ms,0,blend_radius_m)
    movel([0.095014, -1.343433, -2.592257, -0.776698, 1.570796, 1.665810],accel_mss,speed_ms,0,blend_radius_m)
    movel([0.097652, -1.342538, -2.592843, -0.777007, 1.570796, 1.668448],accel_mss,speed_ms,0,blend_radius_m)
    movel([0.099954, -1.341436, -2.593563, -0.777390, 1.570796, 1.670750],accel_mss,speed_ms,0,blend_radius_m)
    movel([0.101868, -1.340096, -2.594436, -0.777857, 1.570796, 1.672665],accel_mss,speed_ms,0,blend_radius_m)
    movel([0.103355, -1.338484, -2.595484, -0.778422, 1.570796, 1.674151],accel_mss,speed_ms,0,blend_radius_m)
    movel([0.104366, -1.336568, -2.596724, -0.779098, 1.570796, 1.675162],accel_mss,speed_ms,0,blend_radius_m)
    movel([0.104758, -1.335128, -2.597652, -0.779609, 1.570796, 1.675554],accel_mss,speed_ms,0,blend_radius_m)
    movel([0.104856, -1.333820, -2.598493, -0.780076, 1.570796, 1.675652],accel_mss,speed_ms,0,blend_radius_m)
    movel([0.104290, -1.331553, -2.599945, -0.780891, 1.570796, 1.675086],accel_mss,speed_ms,0,blend_radius_m)
    movel([0.102903, -1.329680, -2.601140, -0.781569, 1.570796, 1.673699],accel_mss,speed_ms,0,blend_radius_m)
    movel([0.100927, -1.328110, -2.602138, -0.782142, 1.570796, 1.671723],accel_mss,speed_ms,0,blend_radius_m)
    movel([0.096181, -1.325513, -2.603780, -0.783096, 1.570796, 1.666977],accel_mss,speed_ms,0,blend_radius_m)
    movel([0.093898, -1.324290, -2.604551, -0.783548, 1.570796, 1.664694],accel_mss,speed_ms,0,blend_radius_m)
    movel([0.091997, -1.322983, -2.605373, -0.784034, 1.570796, 1.662794],accel_mss,speed_ms,0,blend_radius_m)
    movel([0.089802, -1.320439, -2.606964, -0.784985, 1.570796, 1.660599],accel_mss,speed_ms,0,blend_radius_m)
    movel([0.087728, -1.316904, -2.609163, -0.786322, 1.570796, 1.658524],accel_mss,speed_ms,0,blend_radius_m)
    movel([0.086097, -1.313038, -2.611548, -0.787803, 1.570796, 1.656893],accel_mss,speed_ms,0,blend_radius_m)
    movel([0.085243, -1.309522, -2.613700, -0.789167, 1.570796, 1.656039],accel_mss,speed_ms,0,blend_radius_m)
    movel([0.085334, -1.307066, -2.615193, -0.790129, 1.570796, 1.656131],accel_mss,speed_ms,0,blend_radius_m)
    movel([0.085765, -1.303943, -2.617082, -0.791365, 1.570796, 1.656562],accel_mss,speed_ms,0,blend_radius_m)
    movel([0.086140, -1.300982, -2.618860, -0.792547, 1.570796, 1.656936],accel_mss,speed_ms,0,blend_radius_m)
    movel([0.086054, -1.299040, -2.620020, -0.793329, 1.570796, 1.656850],accel_mss,speed_ms,0,blend_radius_m)
    movel([0.084960, -1.297567, -2.620897, -0.793925, 1.570796, 1.655756],accel_mss,speed_ms,0,blend_radius_m)
    movel([0.083229, -1.296149, -2.621738, -0.794502, 1.570796, 1.654025],accel_mss,speed_ms,0,blend_radius_m)
    movel([0.081337, -1.294543, -2.622688, -0.795158, 1.570796, 1.652133],accel_mss,speed_ms,0,blend_radius_m)
    movel([0.079762, -1.292512, -2.623884, -0.795993, 1.570796, 1.650558],accel_mss,speed_ms,0,blend_radius_m)
    movel([0.079276, -1.291022, -2.624759, -0.796608, 1.570796, 1.650073],accel_mss,speed_ms,0,blend_radius_m)
    speed_ms = 0.003
    movel([0.079276, -1.284127, -2.621447, -0.806816, 1.570796, 1.650073],accel_mss,speed_ms,0,blend_radius_m)
    speed_ms = 0.05
    movel([0.079276, -1.257744, -2.607923, -0.846722, 1.570796, 1.650073],accel_mss,speed_ms,0,blend_radius_m)
    #M_RunCode9
    movel([0.008935, -1.362749, -2.542314, -0.807325, 1.570796, 1.579731],accel_mss,speed_ms,0,blend_radius_m)
    #M_RunCode3
    movel([0.008935, -1.387441, -2.554480, -0.770468, 1.570796, 1.579731],accel_mss,speed_ms,0,blend_radius_m)
    speed_ms = 0.003
    movel([0.008935, -1.393849, -2.557449, -0.761091, 1.570796, 1.579731],accel_mss,speed_ms,0,blend_radius_m)
    speed_ms = 0.02
    movel([0.002258, -1.395296, -2.556397, -0.760696, 1.570796, 1.573054],accel_mss,speed_ms,0,blend_radius_m)
    movel([-0.004092, -1.397246, -2.554974, -0.760170, 1.570796, 1.566704],accel_mss,speed_ms,0,blend_radius_m)
    movel([-0.010095, -1.399609, -2.553241, -0.759539, 1.570796, 1.560701],accel_mss,speed_ms,0,blend_radius_m)
    movel([-0.015722, -1.402293, -2.551264, -0.758832, 1.570796, 1.555074],accel_mss,speed_ms,0,blend_radius_m)
    movel([-0.020960, -1.405211, -2.549103, -0.758076, 1.570796, 1.549836],accel_mss,speed_ms,0,blend_radius_m)
    movel([-0.025788, -1.408280, -2.546815, -0.757294, 1.570796, 1.545008],accel_mss,speed_ms,0,blend_radius_m)
    movel([-0.030195, -1.411415, -2.544465, -0.756509, 1.570796, 1.540602],accel_mss,speed_ms,0,blend_radius_m)
    movel([-0.034169, -1.414536, -2.542110, -0.755742, 1.570796, 1.536627],accel_mss,speed_ms,0,blend_radius_m)
    movel([-0.037701, -1.417563, -2.539813, -0.755013, 1.570796, 1.533095],accel_mss,speed_ms,0,blend_radius_m)
    movel([-0.040785, -1.420426, -2.537628, -0.754335, 1.570796, 1.530011],accel_mss,speed_ms,0,blend_radius_m)
    movel([-0.045575, -1.425346, -2.533844, -0.753199, 1.570796, 1.525221],accel_mss,speed_ms,0,blend_radius_m)
    movel([-0.048490, -1.428716, -2.531231, -0.752442, 1.570796, 1.522306],accel_mss,speed_ms,0,blend_radius_m)
    movel([-0.049477, -1.429967, -2.530257, -0.752165, 1.570796, 1.521319],accel_mss,speed_ms,0,blend_radius_m)
    movel([-0.051122, -1.431920, -2.528731, -0.751738, 1.570796, 1.519674],accel_mss,speed_ms,0,blend_radius_m)
    movel([-0.055029, -1.437224, -2.524558, -0.750606, 1.570796, 1.515767],accel_mss,speed_ms,0,blend_radius_m)
    movel([-0.057348, -1.440864, -2.521671, -0.749854, 1.570796, 1.513448],accel_mss,speed_ms,0,blend_radius_m)
    movel([-0.059655, -1.445019, -2.518349, -0.749020, 1.570796, 1.511141],accel_mss,speed_ms,0,blend_radius_m)
    movel([-0.061765, -1.449583, -2.514671, -0.748135, 1.570796, 1.509031],accel_mss,speed_ms,0,blend_radius_m)
    movel([-0.063497, -1.454451, -2.510713, -0.747225, 1.570796, 1.507299],accel_mss,speed_ms,0,blend_radius_m)
    movel([-0.064672, -1.459521, -2.506551, -0.746316, 1.570796, 1.506124],accel_mss,speed_ms,0,blend_radius_m)
    movel([-0.065124, -1.464696, -2.502263, -0.745429, 1.570796, 1.505673],accel_mss,speed_ms,0,blend_radius_m)
    movel([-0.065026, -1.467294, -2.500095, -0.745000, 1.570796, 1.505770],accel_mss,speed_ms,0,blend_radius_m)
    movel([-0.064684, -1.469882, -2.497925, -0.744582, 1.570796, 1.506112],accel_mss,speed_ms,0,blend_radius_m)
    movel([-0.064082, -1.472455, -2.495757, -0.744177, 1.570796, 1.506714],accel_mss,speed_ms,0,blend_radius_m)
    movel([-0.063198, -1.474997, -2.493605, -0.743787, 1.570796, 1.507598],accel_mss,speed_ms,0,blend_radius_m)
    movel([-0.062011, -1.477502, -2.491475, -0.743412, 1.570796, 1.508785],accel_mss,speed_ms,0,blend_radius_m)
    movel([-0.060507, -1.479958, -2.489377, -0.743054, 1.570796, 1.510289],accel_mss,speed_ms,0,blend_radius_m)
    movel([-0.058664, -1.482358, -2.487317, -0.742714, 1.570796, 1.512132],accel_mss,speed_ms,0,blend_radius_m)
    movel([-0.056462, -1.484695, -2.485303, -0.742391, 1.570796, 1.514334],accel_mss,speed_ms,0,blend_radius_m)
    movel([-0.053886, -1.486960, -2.483343, -0.742086, 1.570796, 1.516910],accel_mss,speed_ms,0,blend_radius_m)
    movel([-0.050917, -1.489148, -2.481442, -0.741799, 1.570796, 1.519879],accel_mss,speed_ms,0,blend_radius_m)
    movel([-0.047538, -1.491249, -2.479610, -0.741531, 1.570796, 1.523258],accel_mss,speed_ms,0,blend_radius_m)
    movel([-0.043727, -1.493261, -2.477848, -0.741280, 1.570796, 1.527070],accel_mss,speed_ms,0,blend_radius_m)
    movel([-0.043413, -1.493399, -2.477727, -0.741263, 1.570796, 1.527384],accel_mss,speed_ms,0,blend_radius_m)
    movel([-0.039203, -1.494916, -2.476395, -0.741078, 1.570796, 1.531593],accel_mss,speed_ms,0,blend_radius_m)
    movel([-0.035098, -1.496113, -2.475341, -0.740935, 1.570796, 1.535698],accel_mss,speed_ms,0,blend_radius_m)
    movel([-0.031097, -1.497007, -2.474552, -0.740830, 1.570796, 1.539699],accel_mss,speed_ms,0,blend_radius_m)
    movel([-0.027200, -1.497619, -2.474012, -0.740759, 1.570796, 1.543596],accel_mss,speed_ms,0,blend_radius_m)
    movel([-0.023401, -1.497961, -2.473709, -0.740719, 1.570796, 1.547395],accel_mss,speed_ms,0,blend_radius_m)
    movel([-0.019703, -1.498054, -2.473627, -0.740708, 1.570796, 1.551094],accel_mss,speed_ms,0,blend_radius_m)
    movel([-0.016102, -1.497914, -2.473750, -0.740724, 1.570796, 1.554694],accel_mss,speed_ms,0,blend_radius_m)
    movel([-0.012603, -1.497558, -2.474065, -0.740766, 1.570796, 1.558193],accel_mss,speed_ms,0,blend_radius_m)
    movel([-0.009202, -1.497002, -2.474557, -0.740831, 1.570796, 1.561594],accel_mss,speed_ms,0,blend_radius_m)
    movel([-0.005904, -1.496264, -2.475207, -0.740918, 1.570796, 1.564892],accel_mss,speed_ms,0,blend_radius_m)
    movel([-0.002707, -1.495360, -2.476004, -0.741025, 1.570796, 1.568089],accel_mss,speed_ms,0,blend_radius_m)
    movel([0.000384, -1.494308, -2.476929, -0.741152, 1.570796, 1.571180],accel_mss,speed_ms,0,blend_radius_m)
    movel([0.006241, -1.491831, -2.479100, -0.741457, 1.570796, 1.577038],accel_mss,speed_ms,0,blend_radius_m)
    movel([0.011644, -1.488969, -2.481598, -0.741822, 1.570796, 1.582441],accel_mss,speed_ms,0,blend_radius_m)
    movel([0.016567, -1.485868, -2.484289, -0.742232, 1.570796, 1.587363],accel_mss,speed_ms,0,blend_radius_m)
    movel([0.020971, -1.482673, -2.487047, -0.742670, 1.570796, 1.591768],accel_mss,speed_ms,0,blend_radius_m)
    movel([0.024820, -1.479535, -2.489739, -0.743115, 1.570796, 1.595617],accel_mss,speed_ms,0,blend_radius_m)
    movel([0.028073, -1.476607, -2.492237, -0.743545, 1.570796, 1.598869],accel_mss,speed_ms,0,blend_radius_m)
    movel([0.032600, -1.472022, -2.496122, -0.744244, 1.570796, 1.603397],accel_mss,speed_ms,0,blend_radius_m)
    movel([0.034188, -1.470205, -2.497653, -0.744530, 1.570796, 1.604984],accel_mss,speed_ms,0,blend_radius_m)
    movel([0.035184, -1.469124, -2.498562, -0.744703, 1.570796, 1.605981],accel_mss,speed_ms,0,blend_radius_m)
    movel([0.037787, -1.466057, -2.501129, -0.745203, 1.570796, 1.608583],accel_mss,speed_ms,0,blend_radius_m)
    movel([0.041425, -1.461251, -2.505123, -0.746015, 1.570796, 1.612221],accel_mss,speed_ms,0,blend_radius_m)
    movel([0.045525, -1.454944, -2.510310, -0.747135, 1.570796, 1.616322],accel_mss,speed_ms,0,blend_radius_m)
    movel([0.047566, -1.451301, -2.513278, -0.747810, 1.570796, 1.618362],accel_mss,speed_ms,0,blend_radius_m)
    movel([0.049501, -1.447374, -2.516456, -0.748560, 1.570796, 1.620297],accel_mss,speed_ms,0,blend_radius_m)
    movel([0.051253, -1.443187, -2.519817, -0.749385, 1.570796, 1.622050],accel_mss,speed_ms,0,blend_radius_m)
    movel([0.052745, -1.438773, -2.523332, -0.750284, 1.570796, 1.623541],accel_mss,speed_ms,0,blend_radius_m)
    movel([0.053894, -1.434165, -2.526970, -0.751254, 1.570796, 1.624690],accel_mss,speed_ms,0,blend_radius_m)
    movel([0.054619, -1.429393, -2.530704, -0.752292, 1.570796, 1.625415],accel_mss,speed_ms,0,blend_radius_m)
    movel([0.054835, -1.424493, -2.534502, -0.753394, 1.570796, 1.625632],accel_mss,speed_ms,0,blend_radius_m)
    movel([0.054448, -1.419502, -2.538335, -0.754553, 1.570796, 1.625244],accel_mss,speed_ms,0,blend_radius_m)
    speed_ms = 0.003
    movel([0.054448, -1.413232, -2.535448, -0.763709, 1.570796, 1.625244],accel_mss,speed_ms,0,blend_radius_m)
    speed_ms = 0.05
    movel([0.054448, -1.389035, -2.523611, -0.799742, 1.570796, 1.625244],accel_mss,speed_ms,0,blend_radius_m)
    #M_RunCode9
    movel([0.026201, -1.394931, -2.519285, -0.798173, 1.570796, 1.596998],accel_mss,speed_ms,0,blend_radius_m)
    #M_RunCode3
    # logo 1
    movel([0.026201, -1.419014, -2.531048, -0.762327, 1.570796, 1.596998],accel_mss,speed_ms,0,blend_radius_m)
    speed_ms = 0.003
    movel([0.026201, -1.425252, -2.533916, -0.753221, 1.570796, 1.596998],accel_mss,speed_ms,0,blend_radius_m)
    speed_ms = 0.007
    movel([0.025327, -1.427673, -2.532041, -0.752675, 1.570796, 1.596124],accel_mss,speed_ms,0,blend_radius_m)
    movel([0.023998, -1.430030, -2.530208, -0.752152, 1.570796, 1.594794],accel_mss,speed_ms,0,blend_radius_m)
    movel([0.022270, -1.432259, -2.528466, -0.751664, 1.570796, 1.593067],accel_mss,speed_ms,0,blend_radius_m)
    movel([0.020204, -1.434300, -2.526864, -0.751225, 1.570796, 1.591001],accel_mss,speed_ms,0,blend_radius_m)
    movel([0.017855, -1.436093, -2.525452, -0.750844, 1.570796, 1.588651],accel_mss,speed_ms,0,blend_radius_m)
    movel([0.015277, -1.437579, -2.524278, -0.750532, 1.570796, 1.586074],accel_mss,speed_ms,0,blend_radius_m)
    movel([0.012524, -1.438697, -2.523392, -0.750300, 1.570796, 1.583320],accel_mss,speed_ms,0,blend_radius_m)
    movel([0.012482, -1.438709, -2.523383, -0.750297, 1.570796, 1.583279],accel_mss,speed_ms,0,blend_radius_m)
    movel([0.006330, -1.440714, -2.521790, -0.749885, 1.570796, 1.577126],accel_mss,speed_ms,0,blend_radius_m)
    movel([0.006274, -1.448361, -2.515659, -0.748369, 1.570796, 1.577070],accel_mss,speed_ms,0,blend_radius_m)
    movel([-0.001028, -1.450748, -2.513727, -0.747914, 1.570796, 1.569769],accel_mss,speed_ms,0,blend_radius_m)
    movel([-0.001057, -1.429246, -2.530818, -0.752325, 1.570796, 1.569739],accel_mss,speed_ms,0,blend_radius_m)
    movel([0.006443, -1.426718, -2.532782, -0.752889, 1.570796, 1.577239],accel_mss,speed_ms,0,blend_radius_m)
    movel([0.006380, -1.434512, -2.526697, -0.751180, 1.570796, 1.577176],accel_mss,speed_ms,0,blend_radius_m)
    movel([0.012652, -1.432447, -2.528318, -0.751624, 1.570796, 1.583448],accel_mss,speed_ms,0,blend_radius_m)
    movel([0.013897, -1.431934, -2.528720, -0.751735, 1.570796, 1.584693],accel_mss,speed_ms,0,blend_radius_m)
    movel([0.015069, -1.431248, -2.529257, -0.751884, 1.570796, 1.585866],accel_mss,speed_ms,0,blend_radius_m)
    movel([0.016140, -1.430418, -2.529905, -0.752066, 1.570796, 1.586937],accel_mss,speed_ms,0,blend_radius_m)
    movel([0.017084, -1.429478, -2.530637, -0.752273, 1.570796, 1.587880],accel_mss,speed_ms,0,blend_radius_m)
    movel([0.017872, -1.428454, -2.531435, -0.752500, 1.570796, 1.588668],accel_mss,speed_ms,0,blend_radius_m)
    movel([0.018477, -1.427379, -2.532270, -0.752740, 1.570796, 1.589274],accel_mss,speed_ms,0,blend_radius_m)
    movel([0.018871, -1.426281, -2.533120, -0.752987, 1.570796, 1.589667],accel_mss,speed_ms,0,blend_radius_m)
    movel([0.019027, -1.425196, -2.533959, -0.753233, 1.570796, 1.589823],accel_mss,speed_ms,0,blend_radius_m)
    movel([0.018923, -1.424191, -2.534735, -0.753463, 1.570796, 1.589719],accel_mss,speed_ms,0,blend_radius_m)
    movel([0.018582, -1.423324, -2.535403, -0.753662, 1.570796, 1.589378],accel_mss,speed_ms,0,blend_radius_m)
    movel([0.017279, -1.422078, -2.536361, -0.753950, 1.570796, 1.588076],accel_mss,speed_ms,0,blend_radius_m)
    movel([0.016369, -1.421728, -2.536630, -0.754031, 1.570796, 1.587166],accel_mss,speed_ms,0,blend_radius_m)
    movel([0.015317, -1.421581, -2.536743, -0.754065, 1.570796, 1.586113],accel_mss,speed_ms,0,blend_radius_m)
    movel([0.014149, -1.421654, -2.536686, -0.754048, 1.570796, 1.584945],accel_mss,speed_ms,0,blend_radius_m)
    movel([0.012893, -1.421962, -2.536451, -0.753977, 1.570796, 1.583690],accel_mss,speed_ms,0,blend_radius_m)
    movel([-0.011765, -1.430336, -2.529969, -0.752084, 1.570796, 1.559031],accel_mss,speed_ms,0,blend_radius_m)
    movel([-0.012922, -1.428926, -2.531068, -0.752396, 1.570796, 1.557874],accel_mss,speed_ms,0,blend_radius_m)
    movel([-0.014385, -1.427793, -2.531948, -0.752648, 1.570796, 1.556411],accel_mss,speed_ms,0,blend_radius_m)
    movel([-0.016128, -1.426956, -2.532598, -0.752835, 1.570796, 1.554668],accel_mss,speed_ms,0,blend_radius_m)
    movel([-0.018121, -1.426429, -2.533006, -0.752954, 1.570796, 1.552676],accel_mss,speed_ms,0,blend_radius_m)
    movel([0.012881, -1.415746, -2.541194, -0.755449, 1.570796, 1.583677],accel_mss,speed_ms,0,blend_radius_m)
    movel([0.015703, -1.415041, -2.541728, -0.755620, 1.570796, 1.586499],accel_mss,speed_ms,0,blend_radius_m)
    movel([0.018324, -1.414849, -2.541874, -0.755666, 1.570796, 1.589120],accel_mss,speed_ms,0,blend_radius_m)
    movel([0.020682, -1.415146, -2.541649, -0.755594, 1.570796, 1.591478],accel_mss,speed_ms,0,blend_radius_m)
    movel([0.022717, -1.415901, -2.541076, -0.755412, 1.570796, 1.593513],accel_mss,speed_ms,0,blend_radius_m)
    movel([0.024378, -1.417079, -2.540181, -0.755129, 1.570796, 1.595175],accel_mss,speed_ms,0,blend_radius_m)
    movel([0.025605, -1.418648, -2.538986, -0.754755, 1.570796, 1.596402],accel_mss,speed_ms,0,blend_radius_m)
    movel([0.026351, -1.420577, -2.537512, -0.754300, 1.570796, 1.597147],accel_mss,speed_ms,0,blend_radius_m)
    movel([0.026558, -1.422828, -2.535785, -0.753776, 1.570796, 1.597354],accel_mss,speed_ms,0,blend_radius_m)
    movel([0.026201, -1.425252, -2.533916, -0.753221, 1.570796, 1.596998],accel_mss,speed_ms,0,blend_radius_m)
    speed_ms = 0.003
    movel([0.026201, -1.419014, -2.531048, -0.762327, 1.570796, 1.596998],accel_mss,speed_ms,0,blend_radius_m)
    speed_ms = 0.05
    movel([0.026201, -1.394931, -2.519285, -0.798173, 1.570796, 1.596998],accel_mss,speed_ms,0,blend_radius_m)
    #M_RunCode9
    movel([0.026290, -1.400953, -2.514815, -0.796621, 1.570796, 1.597086],accel_mss,speed_ms,0,blend_radius_m)
    #M_RunCode3
    # logo 2
    movel([0.026290, -1.424918, -2.526504, -0.760967, 1.570796, 1.597086],accel_mss,speed_ms,0,blend_radius_m)
    speed_ms = 0.003
    movel([0.026290, -1.431124, -2.529354, -0.751912, 1.570796, 1.597086],accel_mss,speed_ms,0,blend_radius_m)
    speed_ms = 0.007
    movel([0.025516, -1.456191, -2.509289, -0.746909, 1.570796, 1.596312],accel_mss,speed_ms,0,blend_radius_m)
    movel([0.025174, -1.458502, -2.507392, -0.746496, 1.570796, 1.595971],accel_mss,speed_ms,0,blend_radius_m)
    movel([0.024333, -1.460806, -2.505491, -0.746092, 1.570796, 1.595129],accel_mss,speed_ms,0,blend_radius_m)
    movel([0.023051, -1.463045, -2.503636, -0.745708, 1.570796, 1.593847],accel_mss,speed_ms,0,blend_radius_m)
    movel([0.021386, -1.465160, -2.501877, -0.745352, 1.570796, 1.592183],accel_mss,speed_ms,0,blend_radius_m)
    movel([0.019396, -1.467090, -2.500266, -0.745033, 1.570796, 1.590192],accel_mss,speed_ms,0,blend_radius_m)
    movel([0.017132, -1.468778, -2.498852, -0.744759, 1.570796, 1.587928],accel_mss,speed_ms,0,blend_radius_m)
    movel([0.014653, -1.470169, -2.497684, -0.744536, 1.570796, 1.585450],accel_mss,speed_ms,0,blend_radius_m)
    movel([0.012007, -1.471206, -2.496811, -0.744372, 1.570796, 1.582804],accel_mss,speed_ms,0,blend_radius_m)
    movel([0.009368, -1.471811, -2.496300, -0.744277, 1.570796, 1.580164],accel_mss,speed_ms,0,blend_radius_m)
    movel([0.006914, -1.471955, -2.496179, -0.744255, 1.570796, 1.577711],accel_mss,speed_ms,0,blend_radius_m)
    movel([0.004695, -1.471666, -2.496423, -0.744300, 1.570796, 1.575491],accel_mss,speed_ms,0,blend_radius_m)
    movel([0.002761, -1.470966, -2.497013, -0.744410, 1.570796, 1.573558],accel_mss,speed_ms,0,blend_radius_m)
    movel([0.001165, -1.469882, -2.497925, -0.744582, 1.570796, 1.571962],accel_mss,speed_ms,0,blend_radius_m)
    movel([-0.000045, -1.468439, -2.499137, -0.744814, 1.570796, 1.570751],accel_mss,speed_ms,0,blend_radius_m)
    movel([-0.000812, -1.466656, -2.500629, -0.745104, 1.570796, 1.569985],accel_mss,speed_ms,0,blend_radius_m)
    movel([-0.001081, -1.464556, -2.502381, -0.745453, 1.570796, 1.569716],accel_mss,speed_ms,0,blend_radius_m)
    movel([-0.001081, -1.464528, -2.502404, -0.745457, 1.570796, 1.569716],accel_mss,speed_ms,0,blend_radius_m)
    movel([-0.001087, -1.459616, -2.506474, -0.746300, 1.570796, 1.569709],accel_mss,speed_ms,0,blend_radius_m)
    movel([-0.010177, -1.462609, -2.503998, -0.745782, 1.570796, 1.560619],accel_mss,speed_ms,0,blend_radius_m)
    movel([-0.010249, -1.456700, -2.508872, -0.746817, 1.570796, 1.560547],accel_mss,speed_ms,0,blend_radius_m)
    movel([0.015495, -1.448305, -2.515704, -0.748379, 1.570796, 1.586292],accel_mss,speed_ms,0,blend_radius_m)
    movel([0.015385, -1.454329, -2.510812, -0.747247, 1.570796, 1.586182],accel_mss,speed_ms,0,blend_radius_m)
    movel([0.006236, -1.457240, -2.508429, -0.746720, 1.570796, 1.577033],accel_mss,speed_ms,0,blend_radius_m)
    movel([0.006199, -1.462239, -2.504305, -0.745845, 1.570796, 1.576995],accel_mss,speed_ms,0,blend_radius_m)
    movel([0.006316, -1.463187, -2.503518, -0.745684, 1.570796, 1.577112],accel_mss,speed_ms,0,blend_radius_m)
    movel([0.006661, -1.464001, -2.502842, -0.745546, 1.570796, 1.577458],accel_mss,speed_ms,0,blend_radius_m)
    movel([0.007215, -1.464664, -2.502290, -0.745435, 1.570796, 1.578011],accel_mss,speed_ms,0,blend_radius_m)
    movel([0.007947, -1.465167, -2.501871, -0.745351, 1.570796, 1.578743],accel_mss,speed_ms,0,blend_radius_m)
    movel([0.008833, -1.465494, -2.501599, -0.745296, 1.570796, 1.579629],accel_mss,speed_ms,0,blend_radius_m)
    movel([0.009848, -1.465633, -2.501483, -0.745273, 1.570796, 1.580644],accel_mss,speed_ms,0,blend_radius_m)
    movel([0.010966, -1.465571, -2.501534, -0.745283, 1.570796, 1.581762],accel_mss,speed_ms,0,blend_radius_m)
    movel([0.012161, -1.465297, -2.501763, -0.745329, 1.570796, 1.582957],accel_mss,speed_ms,0,blend_radius_m)
    movel([0.013362, -1.464825, -2.502156, -0.745408, 1.570796, 1.584158],accel_mss,speed_ms,0,blend_radius_m)
    movel([0.014490, -1.464191, -2.502684, -0.745514, 1.570796, 1.585286],accel_mss,speed_ms,0,blend_radius_m)
    movel([0.016436, -1.462541, -2.504054, -0.745794, 1.570796, 1.587232],accel_mss,speed_ms,0,blend_radius_m)
    movel([0.017199, -1.461582, -2.504849, -0.745958, 1.570796, 1.587995],accel_mss,speed_ms,0,blend_radius_m)
    movel([0.017784, -1.460568, -2.505687, -0.746133, 1.570796, 1.588580],accel_mss,speed_ms,0,blend_radius_m)
    movel([0.018163, -1.459532, -2.506543, -0.746314, 1.570796, 1.588959],accel_mss,speed_ms,0,blend_radius_m)
    movel([0.018312, -1.458496, -2.507396, -0.746497, 1.570796, 1.589108],accel_mss,speed_ms,0,blend_radius_m)
    movel([0.018769, -1.438610, -2.523461, -0.750318, 1.570796, 1.589565],accel_mss,speed_ms,0,blend_radius_m)
    movel([0.020967, -1.436991, -2.524743, -0.750655, 1.570796, 1.591763],accel_mss,speed_ms,0,blend_radius_m)
    movel([0.022974, -1.435181, -2.526171, -0.751037, 1.570796, 1.593771],accel_mss,speed_ms,0,blend_radius_m)
    movel([0.024759, -1.433214, -2.527717, -0.751458, 1.570796, 1.595556],accel_mss,speed_ms,0,blend_radius_m)
    movel([0.026290, -1.431124, -2.529354, -0.751912, 1.570796, 1.597086],accel_mss,speed_ms,0,blend_radius_m)
    speed_ms = 0.003
    movel([0.026290, -1.424918, -2.526504, -0.760967, 1.570796, 1.597086],accel_mss,speed_ms,0,blend_radius_m)
    speed_ms = 0.05
    movel([0.026290, -1.400953, -2.514815, -0.796621, 1.570796, 1.597086],accel_mss,speed_ms,0,blend_radius_m)
    #M_RunCode9
    movel([-0.013828, -1.420647, -2.499837, -0.791905, 1.570796, 1.556968],accel_mss,speed_ms,0,blend_radius_m)
    #M_RunCode3
    # logo 3
    movel([-0.013828, -1.444221, -2.511286, -0.756883, 1.570796, 1.556968],accel_mss,speed_ms,0,blend_radius_m)
    speed_ms = 0.003
    movel([-0.013828, -1.450318, -2.514076, -0.747995, 1.570796, 1.556968],accel_mss,speed_ms,0,blend_radius_m)
    speed_ms = 0.007
    movel([-0.013476, -1.471136, -2.496869, -0.744383, 1.570796, 1.557321],accel_mss,speed_ms,0,blend_radius_m)
    movel([-0.020588, -1.473512, -2.494864, -0.744013, 1.570796, 1.550209],accel_mss,speed_ms,0,blend_radius_m)
    movel([-0.020765, -1.466189, -2.501019, -0.745181, 1.570796, 1.550032],accel_mss,speed_ms,0,blend_radius_m)
    movel([-0.026783, -1.468243, -2.499301, -0.744845, 1.570796, 1.544013],accel_mss,speed_ms,0,blend_radius_m)
    movel([-0.027974, -1.468753, -2.498873, -0.744763, 1.570796, 1.542823],accel_mss,speed_ms,0,blend_radius_m)
    movel([-0.029080, -1.469424, -2.498310, -0.744655, 1.570796, 1.541716],accel_mss,speed_ms,0,blend_radius_m)
    movel([-0.030076, -1.470225, -2.497636, -0.744527, 1.570796, 1.540720],accel_mss,speed_ms,0,blend_radius_m)
    movel([-0.030940, -1.471126, -2.496878, -0.744385, 1.570796, 1.539857],accel_mss,speed_ms,0,blend_radius_m)
    movel([-0.031644, -1.472097, -2.496059, -0.744233, 1.570796, 1.539152],accel_mss,speed_ms,0,blend_radius_m)
    movel([-0.032167, -1.473107, -2.495206, -0.744076, 1.570796, 1.538629],accel_mss,speed_ms,0,blend_radius_m)
    movel([-0.032482, -1.474128, -2.494342, -0.743919, 1.570796, 1.538315],accel_mss,speed_ms,0,blend_radius_m)
    movel([-0.032564, -1.475128, -2.493494, -0.743767, 1.570796, 1.538233],accel_mss,speed_ms,0,blend_radius_m)
    movel([-0.032407, -1.476046, -2.492715, -0.743629, 1.570796, 1.538389],accel_mss,speed_ms,0,blend_radius_m)
    movel([-0.032033, -1.476827, -2.492050, -0.743512, 1.570796, 1.538763],accel_mss,speed_ms,0,blend_radius_m)
    movel([-0.030721, -1.477933, -2.491108, -0.743349, 1.570796, 1.540075],accel_mss,speed_ms,0,blend_radius_m)
    movel([-0.029835, -1.478231, -2.490853, -0.743305, 1.570796, 1.540962],accel_mss,speed_ms,0,blend_radius_m)
    movel([-0.028827, -1.478345, -2.490756, -0.743288, 1.570796, 1.541969],accel_mss,speed_ms,0,blend_radius_m)
    movel([-0.027724, -1.478261, -2.490827, -0.743301, 1.570796, 1.543072],accel_mss,speed_ms,0,blend_radius_m)
    movel([-0.026545, -1.477962, -2.491082, -0.743344, 1.570796, 1.544251],accel_mss,speed_ms,0,blend_radius_m)
    movel([-0.003291, -1.470249, -2.497616, -0.744523, 1.570796, 1.567506],accel_mss,speed_ms,0,blend_radius_m)
    movel([-0.002208, -1.471621, -2.496461, -0.744307, 1.570796, 1.568588],accel_mss,speed_ms,0,blend_radius_m)
    movel([-0.000842, -1.472735, -2.495521, -0.744133, 1.570796, 1.569955],accel_mss,speed_ms,0,blend_radius_m)
    movel([0.000780, -1.473582, -2.494804, -0.744003, 1.570796, 1.571576],accel_mss,speed_ms,0,blend_radius_m)
    movel([0.002630, -1.474149, -2.494324, -0.743916, 1.570796, 1.573427],accel_mss,speed_ms,0,blend_radius_m)
    movel([-0.026259, -1.483597, -2.486251, -0.742542, 1.570796, 1.544537],accel_mss,speed_ms,0,blend_radius_m)
    movel([-0.028868, -1.484263, -2.485676, -0.742450, 1.570796, 1.541929],accel_mss,speed_ms,0,blend_radius_m)
    movel([-0.031310, -1.484475, -2.485493, -0.742421, 1.570796, 1.539487],accel_mss,speed_ms,0,blend_radius_m)
    movel([-0.033538, -1.484257, -2.485681, -0.742451, 1.570796, 1.537258],accel_mss,speed_ms,0,blend_radius_m)
    movel([-0.035499, -1.483634, -2.486219, -0.742536, 1.570796, 1.535298],accel_mss,speed_ms,0,blend_radius_m)
    movel([-0.037143, -1.482628, -2.487085, -0.742676, 1.570796, 1.533653],accel_mss,speed_ms,0,blend_radius_m)
    movel([-0.038418, -1.481261, -2.488259, -0.742868, 1.570796, 1.532378],accel_mss,speed_ms,0,blend_radius_m)
    movel([-0.039266, -1.479557, -2.489720, -0.743112, 1.570796, 1.531530],accel_mss,speed_ms,0,blend_radius_m)
    movel([-0.039631, -1.477534, -2.491448, -0.743408, 1.570796, 1.531165],accel_mss,speed_ms,0,blend_radius_m)
    movel([-0.039470, -1.475322, -2.493329, -0.743738, 1.570796, 1.531326],accel_mss,speed_ms,0,blend_radius_m)
    movel([-0.038807, -1.473075, -2.495233, -0.744081, 1.570796, 1.531989],accel_mss,speed_ms,0,blend_radius_m)
    movel([-0.037686, -1.470854, -2.497107, -0.744428, 1.570796, 1.533111],accel_mss,speed_ms,0,blend_radius_m)
    movel([-0.036153, -1.468720, -2.498901, -0.744768, 1.570796, 1.534644],accel_mss,speed_ms,0,blend_radius_m)
    movel([-0.034263, -1.466735, -2.500563, -0.745091, 1.570796, 1.536533],accel_mss,speed_ms,0,blend_radius_m)
    movel([-0.032061, -1.464965, -2.502040, -0.745384, 1.570796, 1.538735],accel_mss,speed_ms,0,blend_radius_m)
    movel([-0.029604, -1.463474, -2.503280, -0.745635, 1.570796, 1.541193],accel_mss,speed_ms,0,blend_radius_m)
    movel([-0.026944, -1.462330, -2.504230, -0.745830, 1.570796, 1.543852],accel_mss,speed_ms,0,blend_radius_m)
    movel([-0.026910, -1.462325, -2.504233, -0.745830, 1.570796, 1.543886],accel_mss,speed_ms,0,blend_radius_m)
    movel([-0.020919, -1.460257, -2.505944, -0.746188, 1.570796, 1.549878],accel_mss,speed_ms,0,blend_radius_m)
    movel([-0.021113, -1.452818, -2.512045, -0.747526, 1.570796, 1.549683],accel_mss,speed_ms,0,blend_radius_m)
    movel([-0.013828, -1.450318, -2.514076, -0.747995, 1.570796, 1.556968],accel_mss,speed_ms,0,blend_radius_m)
    speed_ms = 0.003
    movel([-0.013828, -1.444221, -2.511286, -0.756883, 1.570796, 1.556968],accel_mss,speed_ms,0,blend_radius_m)
    speed_ms = 0.05
    movel([-0.013828, -1.420647, -2.499837, -0.791905, 1.570796, 1.556968],accel_mss,speed_ms,0,blend_radius_m)
    #M_RunCode9
    movel([-0.004554, -1.414456, -2.504605, -0.793328, 1.570796, 1.566242],accel_mss,speed_ms,0,blend_radius_m)
    #M_RunCode3
    # logo 4
    movel([-0.004554, -1.438154, -2.516128, -0.758106, 1.570796, 1.566242],accel_mss,speed_ms,0,blend_radius_m)
    speed_ms = 0.003
    movel([-0.004554, -1.444286, -2.518937, -0.749166, 1.570796, 1.566242],accel_mss,speed_ms,0,blend_radius_m)
    speed_ms = 0.007
    movel([-0.030413, -1.453190, -2.511742, -0.747457, 1.570796, 1.540384],accel_mss,speed_ms,0,blend_radius_m)
    movel([-0.030631, -1.447262, -2.516546, -0.748581, 1.570796, 1.540165],accel_mss,speed_ms,0,blend_radius_m)
    movel([-0.021373, -1.443998, -2.519168, -0.749223, 1.570796, 1.549423],accel_mss,speed_ms,0,blend_radius_m)
    movel([-0.021506, -1.438931, -2.523207, -0.750251, 1.570796, 1.549290],accel_mss,speed_ms,0,blend_radius_m)
    movel([-0.021659, -1.437966, -2.523971, -0.750451, 1.570796, 1.549137],accel_mss,speed_ms,0,blend_radius_m)
    movel([-0.022051, -1.437150, -2.524617, -0.750622, 1.570796, 1.548746],accel_mss,speed_ms,0,blend_radius_m)
    movel([-0.022654, -1.436495, -2.525135, -0.750759, 1.570796, 1.548142],accel_mss,speed_ms,0,blend_radius_m)
    movel([-0.023440, -1.436013, -2.525515, -0.750861, 1.570796, 1.547356],accel_mss,speed_ms,0,blend_radius_m)
    movel([-0.024383, -1.435717, -2.525748, -0.750924, 1.570796, 1.546414],accel_mss,speed_ms,0,blend_radius_m)
    movel([-0.025453, -1.435620, -2.525825, -0.750944, 1.570796, 1.545344],accel_mss,speed_ms,0,blend_radius_m)
    movel([-0.026625, -1.435736, -2.525733, -0.750920, 1.570796, 1.544171],accel_mss,speed_ms,0,blend_radius_m)
    movel([-0.027869, -1.436075, -2.525466, -0.750848, 1.570796, 1.542928],accel_mss,speed_ms,0,blend_radius_m)
    movel([-0.029104, -1.436621, -2.525035, -0.750733, 1.570796, 1.541692],accel_mss,speed_ms,0,blend_radius_m)
    movel([-0.030257, -1.437330, -2.524475, -0.750584, 1.570796, 1.540539],accel_mss,speed_ms,0,blend_radius_m)
    movel([-0.032206, -1.439115, -2.523061, -0.750213, 1.570796, 1.538590],accel_mss,speed_ms,0,blend_radius_m)
    movel([-0.032945, -1.440126, -2.522258, -0.750005, 1.570796, 1.537851],accel_mss,speed_ms,0,blend_radius_m)
    movel([-0.033494, -1.441179, -2.521420, -0.749790, 1.570796, 1.537302],accel_mss,speed_ms,0,blend_radius_m)
    movel([-0.033825, -1.442242, -2.520572, -0.749575, 1.570796, 1.536971],accel_mss,speed_ms,0,blend_radius_m)
    movel([-0.033916, -1.443288, -2.519736, -0.749365, 1.570796, 1.536881],accel_mss,speed_ms,0,blend_radius_m)
    movel([-0.033109, -1.462629, -2.503981, -0.745779, 1.570796, 1.537687],accel_mss,speed_ms,0,blend_radius_m)
    movel([-0.035187, -1.464253, -2.502633, -0.745504, 1.570796, 1.535609],accel_mss,speed_ms,0,blend_radius_m)
    movel([-0.037047, -1.466037, -2.501146, -0.745206, 1.570796, 1.533749],accel_mss,speed_ms,0,blend_radius_m)
    movel([-0.038661, -1.467949, -2.499547, -0.744893, 1.570796, 1.532136],accel_mss,speed_ms,0,blend_radius_m)
    movel([-0.040005, -1.469956, -2.497863, -0.744570, 1.570796, 1.530791],accel_mss,speed_ms,0,blend_radius_m)
    movel([-0.041210, -1.446018, -2.517547, -0.748824, 1.570796, 1.529586],accel_mss,speed_ms,0,blend_radius_m)
    movel([-0.041047, -1.443712, -2.519397, -0.749280, 1.570796, 1.529749],accel_mss,speed_ms,0,blend_radius_m)
    movel([-0.040357, -1.441360, -2.521276, -0.749753, 1.570796, 1.530439],accel_mss,speed_ms,0,blend_radius_m)
    movel([-0.039188, -1.439029, -2.523129, -0.750231, 1.570796, 1.531608],accel_mss,speed_ms,0,blend_radius_m)
    movel([-0.037595, -1.436783, -2.524907, -0.750699, 1.570796, 1.533201],accel_mss,speed_ms,0,blend_radius_m)
    movel([-0.035626, -1.434684, -2.526562, -0.751143, 1.570796, 1.535170],accel_mss,speed_ms,0,blend_radius_m)
    movel([-0.033334, -1.432807, -2.528036, -0.751546, 1.570796, 1.537463],accel_mss,speed_ms,0,blend_radius_m)
    movel([-0.030776, -1.431217, -2.529281, -0.751891, 1.570796, 1.540020],accel_mss,speed_ms,0,blend_radius_m)
    movel([-0.028011, -1.429984, -2.530243, -0.752162, 1.570796, 1.542785],accel_mss,speed_ms,0,blend_radius_m)
    movel([-0.025224, -1.429209, -2.530848, -0.752333, 1.570796, 1.545572],accel_mss,speed_ms,0,blend_radius_m)
    movel([-0.022615, -1.428937, -2.531059, -0.752393, 1.570796, 1.548182],accel_mss,speed_ms,0,blend_radius_m)
    movel([-0.020244, -1.429141, -2.530901, -0.752348, 1.570796, 1.550552],accel_mss,speed_ms,0,blend_radius_m)
    movel([-0.018170, -1.429794, -2.530392, -0.752203, 1.570796, 1.552627],accel_mss,speed_ms,0,blend_radius_m)
    movel([-0.016452, -1.430869, -2.529553, -0.751967, 1.570796, 1.554344],accel_mss,speed_ms,0,blend_radius_m)
    movel([-0.015150, -1.432337, -2.528404, -0.751647, 1.570796, 1.555647],accel_mss,speed_ms,0,blend_radius_m)
    movel([-0.014311, -1.434169, -2.526967, -0.751253, 1.570796, 1.556485],accel_mss,speed_ms,0,blend_radius_m)
    movel([-0.013996, -1.436334, -2.525261, -0.750793, 1.570796, 1.556800],accel_mss,speed_ms,0,blend_radius_m)
    movel([-0.013995, -1.436365, -2.525237, -0.750787, 1.570796, 1.556801],accel_mss,speed_ms,0,blend_radius_m)
    movel([-0.013905, -1.441407, -2.521238, -0.749744, 1.570796, 1.556892],accel_mss,speed_ms,0,blend_radius_m)
    movel([-0.004588, -1.438226, -2.523765, -0.750397, 1.570796, 1.566208],accel_mss,speed_ms,0,blend_radius_m)
    movel([-0.004554, -1.444286, -2.518937, -0.749166, 1.570796, 1.566242],accel_mss,speed_ms,0,blend_radius_m)
    speed_ms = 0.003
    movel([-0.004554, -1.438154, -2.516128, -0.758106, 1.570796, 1.566242],accel_mss,speed_ms,0,blend_radius_m)
    speed_ms = 0.05
    movel([-0.004554, -1.414456, -2.504605, -0.793328, 1.570796, 1.566242],accel_mss,speed_ms,0,blend_radius_m)
    #M_RunCode9
    movel([-0.032291, -1.468457, -2.461136, -0.782796, 1.570796, 1.538506],accel_mss,speed_ms,0,blend_radius_m)
    #M_RunCode3
    movel([-0.032291, -1.491047, -2.472019, -0.749323, 1.570796, 1.538506],accel_mss,speed_ms,0,blend_radius_m)
    speed_ms = 0.003
    movel([-0.032291, -1.496876, -2.474668, -0.740846, 1.570796, 1.538506],accel_mss,speed_ms,0,blend_radius_m)
    speed_ms = 0.02
    movel([-0.028289, -1.497853, -2.473805, -0.740732, 1.570796, 1.542507],accel_mss,speed_ms,0,blend_radius_m)
    movel([-0.022483, -1.498634, -2.473113, -0.740642, 1.570796, 1.548314],accel_mss,speed_ms,0,blend_radius_m)
    movel([-0.015478, -1.499183, -2.472627, -0.740579, 1.570796, 1.555318],accel_mss,speed_ms,0,blend_radius_m)
    movel([-0.007866, -1.499452, -2.472389, -0.740548, 1.570796, 1.562930],accel_mss,speed_ms,0,blend_radius_m)
    movel([-0.000234, -1.499375, -2.472457, -0.740557, 1.570796, 1.570562],accel_mss,speed_ms,0,blend_radius_m)
    movel([0.006843, -1.498869, -2.472905, -0.740615, 1.570796, 1.577639],accel_mss,speed_ms,0,blend_radius_m)
    movel([0.009997, -1.498425, -2.473298, -0.740666, 1.570796, 1.580793],accel_mss,speed_ms,0,blend_radius_m)
    movel([0.012799, -1.497838, -2.473818, -0.740733, 1.570796, 1.583595],accel_mss,speed_ms,0,blend_radius_m)
    movel([0.015179, -1.497090, -2.474478, -0.740820, 1.570796, 1.585975],accel_mss,speed_ms,0,blend_radius_m)
    movel([0.017064, -1.496170, -2.475290, -0.740929, 1.570796, 1.587860],accel_mss,speed_ms,0,blend_radius_m)
    movel([0.018305, -1.495130, -2.476206, -0.741053, 1.570796, 1.589102],accel_mss,speed_ms,0,blend_radius_m)
    movel([0.018536, -1.494672, -2.476609, -0.741108, 1.570796, 1.589332],accel_mss,speed_ms,0,blend_radius_m)
    movel([0.018533, -1.494254, -2.476977, -0.741159, 1.570796, 1.589329],accel_mss,speed_ms,0,blend_radius_m)
    movel([0.017910, -1.493516, -2.477625, -0.741249, 1.570796, 1.588706],accel_mss,speed_ms,0,blend_radius_m)
    movel([0.016604, -1.492895, -2.478169, -0.741325, 1.570796, 1.587400],accel_mss,speed_ms,0,blend_radius_m)
    movel([0.012601, -1.491915, -2.479027, -0.741447, 1.570796, 1.583398],accel_mss,speed_ms,0,blend_radius_m)
    movel([0.007868, -1.491121, -2.479721, -0.741547, 1.570796, 1.578664],accel_mss,speed_ms,0,blend_radius_m)
    speed_ms = 0.003
    movel([0.007868, -1.485259, -2.477055, -0.750075, 1.570796, 1.578664],accel_mss,speed_ms,0,blend_radius_m)
    speed_ms = 0.05
    movel([0.007868, -1.462545, -2.466104, -0.783740, 1.570796, 1.578664],accel_mss,speed_ms,0,blend_radius_m)
    #M_RunCode9
    movel([0.111252, -1.362130, -2.542744, -0.807516, 1.570796, 1.682048],accel_mss,speed_ms,0,blend_radius_m)
    #M_RunCode3
    movel([0.111252, -1.386833, -2.554917, -0.770639, 1.570796, 1.682048],accel_mss,speed_ms,0,blend_radius_m)
    speed_ms = 0.003
    movel([0.111252, -1.393244, -2.557888, -0.761257, 1.570796, 1.682048],accel_mss,speed_ms,0,blend_radius_m)
    speed_ms = 0.02
    movel([0.110885, -1.392563, -2.558382, -0.761444, 1.570796, 1.681681],accel_mss,speed_ms,0,blend_radius_m)
    movel([0.111193, -1.391640, -2.559050, -0.761699, 1.570796, 1.681989],accel_mss,speed_ms,0,blend_radius_m)
    movel([0.111430, -1.391289, -2.559304, -0.761796, 1.570796, 1.682226],accel_mss,speed_ms,0,blend_radius_m)
    movel([0.113227, -1.388600, -2.561242, -0.762547, 1.570796, 1.684023],accel_mss,speed_ms,0,blend_radius_m)
    movel([0.114913, -1.385812, -2.563240, -0.763337, 1.570796, 1.685709],accel_mss,speed_ms,0,blend_radius_m)
    movel([0.116248, -1.383009, -2.565238, -0.764142, 1.570796, 1.687044],accel_mss,speed_ms,0,blend_radius_m)
    movel([0.116992, -1.380278, -2.567174, -0.764937, 1.570796, 1.687789],accel_mss,speed_ms,0,blend_radius_m)
    movel([0.116968, -1.377745, -2.568959, -0.765685, 1.570796, 1.687764],accel_mss,speed_ms,0,blend_radius_m)
    movel([0.116316, -1.375443, -2.570574, -0.766372, 1.570796, 1.687112],accel_mss,speed_ms,0,blend_radius_m)
    movel([0.115270, -1.373335, -2.572046, -0.767007, 1.570796, 1.686067],accel_mss,speed_ms,0,blend_radius_m)
    movel([0.114064, -1.371392, -2.573398, -0.767599, 1.570796, 1.684860],accel_mss,speed_ms,0,blend_radius_m)
    movel([0.113890, -1.371125, -2.573583, -0.767681, 1.570796, 1.684687],accel_mss,speed_ms,0,blend_radius_m)
    movel([0.113812, -1.370278, -2.574170, -0.767941, 1.570796, 1.684608],accel_mss,speed_ms,0,blend_radius_m)
    movel([0.114407, -1.369313, -2.574838, -0.768238, 1.570796, 1.685203],accel_mss,speed_ms,0,blend_radius_m)
    movel([0.115418, -1.368629, -2.575310, -0.768450, 1.570796, 1.686215],accel_mss,speed_ms,0,blend_radius_m)
    movel([0.116424, -1.368527, -2.575381, -0.768481, 1.570796, 1.687220],accel_mss,speed_ms,0,blend_radius_m)
    movel([0.116753, -1.368610, -2.575323, -0.768455, 1.570796, 1.687549],accel_mss,speed_ms,0,blend_radius_m)
    movel([0.119272, -1.369228, -2.574897, -0.768264, 1.570796, 1.690068],accel_mss,speed_ms,0,blend_radius_m)
    movel([0.121948, -1.369693, -2.574575, -0.768121, 1.570796, 1.692744],accel_mss,speed_ms,0,blend_radius_m)
    movel([0.124783, -1.369803, -2.574499, -0.768087, 1.570796, 1.695579],accel_mss,speed_ms,0,blend_radius_m)
    movel([0.127781, -1.369353, -2.574810, -0.768226, 1.570796, 1.698577],accel_mss,speed_ms,0,blend_radius_m)
    movel([0.130879, -1.368222, -2.575591, -0.768576, 1.570796, 1.701675],accel_mss,speed_ms,0,blend_radius_m)
    movel([0.133979, -1.366570, -2.576729, -0.769091, 1.570796, 1.704775],accel_mss,speed_ms,0,blend_radius_m)
    movel([0.137021, -1.364614, -2.578070, -0.769705, 1.570796, 1.707817],accel_mss,speed_ms,0,blend_radius_m)
    movel([0.139948, -1.362567, -2.579468, -0.770353, 1.570796, 1.710744],accel_mss,speed_ms,0,blend_radius_m)
    movel([0.140351, -1.362282, -2.579663, -0.770444, 1.570796, 1.711147],accel_mss,speed_ms,0,blend_radius_m)
    movel([0.141415, -1.361842, -2.579963, -0.770585, 1.570796, 1.712211],accel_mss,speed_ms,0,blend_radius_m)
    movel([0.142303, -1.362034, -2.579832, -0.770523, 1.570796, 1.713099],accel_mss,speed_ms,0,blend_radius_m)
    movel([0.142651, -1.362763, -2.579335, -0.770291, 1.570796, 1.713448],accel_mss,speed_ms,0,blend_radius_m)
    movel([0.142301, -1.363732, -2.578674, -0.769984, 1.570796, 1.713097],accel_mss,speed_ms,0,blend_radius_m)
    movel([0.142048, -1.364092, -2.578428, -0.769870, 1.570796, 1.712845],accel_mss,speed_ms,0,blend_radius_m)
    movel([0.140125, -1.366877, -2.576517, -0.768994, 1.570796, 1.710921],accel_mss,speed_ms,0,blend_radius_m)
    movel([0.138331, -1.369745, -2.574539, -0.768105, 1.570796, 1.709127],accel_mss,speed_ms,0,blend_radius_m)
    movel([0.136909, -1.372607, -2.572554, -0.767229, 1.570796, 1.707706],accel_mss,speed_ms,0,blend_radius_m)
    movel([0.136098, -1.375380, -2.570618, -0.766391, 1.570796, 1.706895],accel_mss,speed_ms,0,blend_radius_m)
    movel([0.136067, -1.377942, -2.568821, -0.765626, 1.570796, 1.706863],accel_mss,speed_ms,0,blend_radius_m)
    movel([0.136654, -1.380269, -2.567180, -0.764940, 1.570796, 1.707451],accel_mss,speed_ms,0,blend_radius_m)
    movel([0.137628, -1.382399, -2.565672, -0.764319, 1.570796, 1.708424],accel_mss,speed_ms,0,blend_radius_m)
    movel([0.138754, -1.384367, -2.564272, -0.763751, 1.570796, 1.709550],accel_mss,speed_ms,0,blend_radius_m)
    movel([0.138923, -1.384659, -2.564063, -0.763667, 1.570796, 1.709719],accel_mss,speed_ms,0,blend_radius_m)
    movel([0.138935, -1.384688, -2.564043, -0.763658, 1.570796, 1.709731],accel_mss,speed_ms,0,blend_radius_m)
    movel([0.138981, -1.384800, -2.563963, -0.763626, 1.570796, 1.709777],accel_mss,speed_ms,0,blend_radius_m)
    movel([0.138936, -1.385591, -2.563398, -0.763400, 1.570796, 1.709732],accel_mss,speed_ms,0,blend_radius_m)
    movel([0.138346, -1.386416, -2.562808, -0.763165, 1.570796, 1.709142],accel_mss,speed_ms,0,blend_radius_m)
    movel([0.137483, -1.387016, -2.562379, -0.762994, 1.570796, 1.708279],accel_mss,speed_ms,0,blend_radius_m)
    movel([0.136587, -1.387162, -2.562274, -0.762953, 1.570796, 1.707383],accel_mss,speed_ms,0,blend_radius_m)
    movel([0.136437, -1.387138, -2.562291, -0.762960, 1.570796, 1.707233],accel_mss,speed_ms,0,blend_radius_m)
    movel([0.136409, -1.387135, -2.562294, -0.762961, 1.570796, 1.707205],accel_mss,speed_ms,0,blend_radius_m)
    movel([0.136357, -1.387121, -2.562304, -0.762965, 1.570796, 1.707153],accel_mss,speed_ms,0,blend_radius_m)
    movel([0.136070, -1.387035, -2.562365, -0.762989, 1.570796, 1.706866],accel_mss,speed_ms,0,blend_radius_m)
    movel([0.133632, -1.386368, -2.562842, -0.763178, 1.570796, 1.704428],accel_mss,speed_ms,0,blend_radius_m)
    movel([0.131029, -1.385863, -2.563204, -0.763322, 1.570796, 1.701826],accel_mss,speed_ms,0,blend_radius_m)
    movel([0.128257, -1.385721, -2.563306, -0.763363, 1.570796, 1.699053],accel_mss,speed_ms,0,blend_radius_m)
    movel([0.125317, -1.386137, -2.563008, -0.763244, 1.570796, 1.696114],accel_mss,speed_ms,0,blend_radius_m)
    movel([0.122291, -1.387227, -2.562227, -0.762934, 1.570796, 1.693087],accel_mss,speed_ms,0,blend_radius_m)
    movel([0.119277, -1.388829, -2.561077, -0.762483, 1.570796, 1.690073],accel_mss,speed_ms,0,blend_radius_m)
    movel([0.116340, -1.390726, -2.559711, -0.761952, 1.570796, 1.687136],accel_mss,speed_ms,0,blend_radius_m)
    movel([0.113539, -1.392701, -2.558282, -0.761406, 1.570796, 1.684336],accel_mss,speed_ms,0,blend_radius_m)
    movel([0.113148, -1.392983, -2.558078, -0.761328, 1.570796, 1.683944],accel_mss,speed_ms,0,blend_radius_m)
    movel([0.112540, -1.393306, -2.557843, -0.761239, 1.570796, 1.683337],accel_mss,speed_ms,0,blend_radius_m)
    movel([0.111945, -1.393428, -2.557755, -0.761206, 1.570796, 1.682741],accel_mss,speed_ms,0,blend_radius_m)
    movel([0.111252, -1.393244, -2.557888, -0.761257, 1.570796, 1.682048],accel_mss,speed_ms,0,blend_radius_m)
    speed_ms = 0.003
    movel([0.111252, -1.386833, -2.554917, -0.770639, 1.570796, 1.682048],accel_mss,speed_ms,0,blend_radius_m)
    speed_ms = 0.05
    movel([0.111252, -1.362130, -2.542744, -0.807516, 1.570796, 1.682048],accel_mss,speed_ms,0,blend_radius_m)
    #M_RunCode9
    movel([-0.084369, -1.456146, -2.471422, -0.784820, 1.570796, 1.486428],accel_mss,speed_ms,0,blend_radius_m)
    #M_RunCode3
    movel([-0.084369, -1.478994, -2.482448, -0.750947, 1.570796, 1.486428],accel_mss,speed_ms,0,blend_radius_m)
    speed_ms = 0.003
    movel([-0.084369, -1.484892, -2.485133, -0.742364, 1.570796, 1.486428],accel_mss,speed_ms,0,blend_radius_m)
    speed_ms = 0.02
    movel([-0.084440, -1.485448, -2.484653, -0.742289, 1.570796, 1.486356],accel_mss,speed_ms,0,blend_radius_m)
    movel([-0.084547, -1.485666, -2.484463, -0.742259, 1.570796, 1.486250],accel_mss,speed_ms,0,blend_radius_m)
    movel([-0.086065, -1.489082, -2.481499, -0.741807, 1.570796, 1.484731],accel_mss,speed_ms,0,blend_radius_m)
    movel([-0.086534, -1.490770, -2.480028, -0.741591, 1.570796, 1.484263],accel_mss,speed_ms,0,blend_radius_m)
    movel([-0.086615, -1.492352, -2.478644, -0.741392, 1.570796, 1.484182],accel_mss,speed_ms,0,blend_radius_m)
    movel([-0.086218, -1.493745, -2.477423, -0.741220, 1.570796, 1.484579],accel_mss,speed_ms,0,blend_radius_m)
    movel([-0.085447, -1.494948, -2.476366, -0.741075, 1.570796, 1.485349],accel_mss,speed_ms,0,blend_radius_m)
    movel([-0.083383, -1.496965, -2.474589, -0.740835, 1.570796, 1.487414],accel_mss,speed_ms,0,blend_radius_m)
    movel([-0.083221, -1.497107, -2.474463, -0.740818, 1.570796, 1.487575],accel_mss,speed_ms,0,blend_radius_m)
    movel([-0.083211, -1.497121, -2.474451, -0.740817, 1.570796, 1.487586],accel_mss,speed_ms,0,blend_radius_m)
    movel([-0.083162, -1.497178, -2.474401, -0.740810, 1.570796, 1.487634],accel_mss,speed_ms,0,blend_radius_m)
    movel([-0.083060, -1.497614, -2.474015, -0.740759, 1.570796, 1.487736],accel_mss,speed_ms,0,blend_radius_m)
    movel([-0.083317, -1.498126, -2.473563, -0.740700, 1.570796, 1.487480],accel_mss,speed_ms,0,blend_radius_m)
    movel([-0.083792, -1.498543, -2.473194, -0.740652, 1.570796, 1.487004],accel_mss,speed_ms,0,blend_radius_m)
    movel([-0.084362, -1.498714, -2.473042, -0.740632, 1.570796, 1.486434],accel_mss,speed_ms,0,blend_radius_m)
    movel([-0.084466, -1.498717, -2.473040, -0.740632, 1.570796, 1.486331],accel_mss,speed_ms,0,blend_radius_m)
    movel([-0.084486, -1.498718, -2.473039, -0.740632, 1.570796, 1.486311],accel_mss,speed_ms,0,blend_radius_m)
    movel([-0.084522, -1.498716, -2.473041, -0.740632, 1.570796, 1.486274],accel_mss,speed_ms,0,blend_radius_m)
    movel([-0.084728, -1.498699, -2.473056, -0.740634, 1.570796, 1.486068],accel_mss,speed_ms,0,blend_radius_m)
    movel([-0.088264, -1.498571, -2.473169, -0.740649, 1.570796, 1.482533],accel_mss,speed_ms,0,blend_radius_m)
    movel([-0.090124, -1.498771, -2.472992, -0.740626, 1.570796, 1.480672],accel_mss,speed_ms,0,blend_radius_m)
    movel([-0.092005, -1.499294, -2.472529, -0.740566, 1.570796, 1.478792],accel_mss,speed_ms,0,blend_radius_m)
    movel([-0.093835, -1.500192, -2.471732, -0.740465, 1.570796, 1.476961],accel_mss,speed_ms,0,blend_radius_m)
    movel([-0.095575, -1.501368, -2.470686, -0.740334, 1.570796, 1.475222],accel_mss,speed_ms,0,blend_radius_m)
    movel([-0.098764, -1.504060, -2.468286, -0.740043, 1.570796, 1.472032],accel_mss,speed_ms,0,blend_radius_m)
    movel([-0.098978, -1.504252, -2.468115, -0.740023, 1.570796, 1.471818],accel_mss,speed_ms,0,blend_radius_m)
    movel([-0.099706, -1.504614, -2.467790, -0.739985, 1.570796, 1.471091],accel_mss,speed_ms,0,blend_radius_m)
    movel([-0.100193, -1.504581, -2.467820, -0.739988, 1.570796, 1.470603],accel_mss,speed_ms,0,blend_radius_m)
    movel([-0.100545, -1.504241, -2.468124, -0.740024, 1.570796, 1.470252],accel_mss,speed_ms,0,blend_radius_m)
    movel([-0.100485, -1.503703, -2.468605, -0.740081, 1.570796, 1.470311],accel_mss,speed_ms,0,blend_radius_m)
    movel([-0.100382, -1.503485, -2.468799, -0.740104, 1.570796, 1.470414],accel_mss,speed_ms,0,blend_radius_m)
    movel([-0.098943, -1.500141, -2.471777, -0.740471, 1.570796, 1.471853],accel_mss,speed_ms,0,blend_radius_m)
    movel([-0.098503, -1.498476, -2.473253, -0.740660, 1.570796, 1.472293],accel_mss,speed_ms,0,blend_radius_m)
    movel([-0.098445, -1.496914, -2.474634, -0.740841, 1.570796, 1.472351],accel_mss,speed_ms,0,blend_radius_m)
    movel([-0.098863, -1.495539, -2.475846, -0.741004, 1.570796, 1.471934],accel_mss,speed_ms,0,blend_radius_m)
    movel([-0.099657, -1.494351, -2.476892, -0.741147, 1.570796, 1.471140],accel_mss,speed_ms,0,blend_radius_m)
    movel([-0.101778, -1.492373, -2.478626, -0.741390, 1.570796, 1.469018],accel_mss,speed_ms,0,blend_radius_m)
    movel([-0.101934, -1.492246, -2.478737, -0.741406, 1.570796, 1.468862],accel_mss,speed_ms,0,blend_radius_m)
    movel([-0.102121, -1.491796, -2.479131, -0.741462, 1.570796, 1.468676],accel_mss,speed_ms,0,blend_radius_m)
    movel([-0.101882, -1.491218, -2.479636, -0.741534, 1.570796, 1.468914],accel_mss,speed_ms,0,blend_radius_m)
    movel([-0.101327, -1.490751, -2.480044, -0.741593, 1.570796, 1.469469],accel_mss,speed_ms,0,blend_radius_m)
    movel([-0.100683, -1.490599, -2.480177, -0.741613, 1.570796, 1.470114],accel_mss,speed_ms,0,blend_radius_m)
    movel([-0.100452, -1.490613, -2.480165, -0.741611, 1.570796, 1.470344],accel_mss,speed_ms,0,blend_radius_m)
    movel([-0.096866, -1.490691, -2.480097, -0.741601, 1.570796, 1.473930],accel_mss,speed_ms,0,blend_radius_m)
    movel([-0.094982, -1.490470, -2.480289, -0.741629, 1.570796, 1.475815],accel_mss,speed_ms,0,blend_radius_m)
    movel([-0.093081, -1.489931, -2.480760, -0.741698, 1.570796, 1.477716],accel_mss,speed_ms,0,blend_radius_m)
    movel([-0.091225, -1.489014, -2.481558, -0.741816, 1.570796, 1.479571],accel_mss,speed_ms,0,blend_radius_m)
    movel([-0.089453, -1.487814, -2.482602, -0.741973, 1.570796, 1.481343],accel_mss,speed_ms,0,blend_radius_m)
    movel([-0.086181, -1.485064, -2.484985, -0.742341, 1.570796, 1.484616],accel_mss,speed_ms,0,blend_radius_m)
    movel([-0.085961, -1.484870, -2.485152, -0.742367, 1.570796, 1.484835],accel_mss,speed_ms,0,blend_radius_m)
    movel([-0.085335, -1.484527, -2.485448, -0.742414, 1.570796, 1.485462],accel_mss,speed_ms,0,blend_radius_m)
    movel([-0.084720, -1.484539, -2.485438, -0.742412, 1.570796, 1.486076],accel_mss,speed_ms,0,blend_radius_m)
    movel([-0.084369, -1.484892, -2.485133, -0.742364, 1.570796, 1.486428],accel_mss,speed_ms,0,blend_radius_m)
    speed_ms = 0.003
    movel([-0.084369, -1.478994, -2.482448, -0.750947, 1.570796, 1.486428],accel_mss,speed_ms,0,blend_radius_m)
    speed_ms = 0.05
    movel([-0.084369, -1.456146, -2.471422, -0.784820, 1.570796, 1.486428],accel_mss,speed_ms,0,blend_radius_m)
    #M_RunCode9
    movel([-0.182919, -1.301620, -2.582217, -0.828551, 1.570796, 1.387878],accel_mss,speed_ms,0,blend_radius_m)
    movel([-0.182919, -1.244008, -2.547730, -0.920652, 1.570796, 1.387878],accel_mss,speed_ms,0,blend_radius_m)
    #M_RunCode2
    # End of main program
  end

  Machining1()
end
